C07305=1215.295,-74.617,-38.578,179.642,5.411,149.053
C07306=1215.289,-74.347,-38.590,179.644,5.412,149.052
C07307=1215.284,-74.097,-38.601,179.647,5.412,149.051
C07308=1215.278,-73.847,-38.613,179.649,5.412,149.051
C07309=1215.274,-73.598,-38.625,179.652,5.412,149.050
C07310=1215.268,-73.348,-38.636,179.653,5.412,149.049
C07311=1215.263,-73.098,-38.647,179.656,5.413,149.049
C07312=1215.258,-72.848,-38.658,179.658,5.413,149.048
C07313=1215.253,-72.599,-38.670,179.661,5.413,149.047
C07314=1215.247,-72.350,-38.681,179.663,5.413,149.047
C07315=1215.242,-72.100,-38.693,179.665,5.413,149.046
C07316=1215.237,-71.850,-38.704,179.668,5.414,149.045
C07317=1215.232,-71.600,-38.715,179.670,5.413,149.045
C07318=1215.227,-71.350,-38.726,179.673,5.414,149.044
C07319=1215.221,-71.101,-38.737,179.675,5.413,149.043
C07320=1215.216,-70.851,-38.749,179.677,5.414,149.043
C07321=1215.211,-70.601,-38.760,179.680,5.415,149.042
C07322=1215.206,-70.351,-38.772,179.682,5.414,149.041
C07323=1215.201,-70.103,-38.783,179.685,5.415,149.041
C07324=1215.195,-69.853,-38.795,179.687,5.414,149.040
C07325=1215.190,-69.603,-38.806,179.689,5.415,149.039
C07326=1215.185,-69.353,-38.818,179.691,5.414,149.038
C07327=1215.180,-69.103,-38.829,179.694,5.415,149.038
C07328=1215.174,-68.854,-38.840,179.697,5.415,149.037
C07329=1215.169,-68.604,-38.852,179.699,5.415,149.036
C07330=1215.164,-68.354,-38.864,179.701,5.416,149.036
C07331=1215.159,-68.104,-38.875,179.703,5.415,149.035
C07332=1215.154,-67.854,-38.887,179.706,5.416,149.034
C07333=1215.149,-67.605,-38.898,179.708,5.416,149.034
C07334=1215.143,-67.356,-38.910,179.711,5.416,149.033
C07335=1215.138,-67.106,-38.921,179.713,5.416,149.032
C07336=1215.133,-66.856,-38.933,179.715,5.416,149.032
C07337=1215.128,-66.606,-38.944,179.718,5.417,149.031
C07338=1215.123,-66.356,-38.956,179.720,5.416,149.030
C07339=1215.118,-66.107,-38.967,179.723,5.417,149.029
C07340=1215.112,-65.858,-38.979,179.725,5.416,149.029
C07341=1215.107,-65.608,-38.990,179.727,5.417,149.028
C07342=1215.102,-65.358,-39.002,179.730,5.418,149.028
C07343=1215.097,-65.108,-39.014,179.732,5.417,149.027
C07344=1215.092,-64.858,-39.025,179.734,5.418,149.026
C07345=1215.086,-64.609,-39.037,179.737,5.417,149.025
C07346=1215.082,-64.360,-39.049,179.739,5.418,149.025
C07347=1215.077,-64.110,-39.061,179.741,5.417,149.024
C07348=1215.071,-63.861,-39.072,179.744,5.418,149.023
C07349=1215.066,-63.611,-39.084,179.747,5.418,149.023
C07350=1215.060,-63.361,-39.096,179.749,5.418,149.022
C07351=1215.056,-63.111,-39.107,179.751,5.418,149.021
C07352=1215.050,-62.861,-39.119,179.753,5.418,149.020
C07353=1215.046,-62.612,-39.130,179.756,5.419,149.020
C07354=1215.040,-62.362,-39.142,179.758,5.419,149.019
C07355=1215.035,-62.112,-39.154,179.760,5.419,149.019
C07356=1215.030,-61.863,-39.166,179.763,5.420,149.018
C07357=1215.024,-61.614,-39.177,179.765,5.419,149.017
C07358=1215.019,-61.364,-39.189,179.768,5.420,149.016
C07359=1215.014,-61.114,-39.201,179.770,5.420,149.016
C07360=1215.009,-60.864,-39.212,179.773,5.420,149.015
C07361=1215.003,-60.614,-39.224,179.775,5.420,149.014
C07362=1214.999,-60.365,-39.236,179.777,5.420,149.014
C07363=1214.994,-60.115,-39.248,179.780,5.420,149.013
C07364=1214.988,-59.865,-39.260,179.783,5.421,149.012
C07365=1214.983,-59.616,-39.271,179.784,5.421,149.012
C07366=1214.978,-59.366,-39.283,179.787,5.421,149.011
C07367=1214.973,-59.116,-39.296,179.789,5.421,149.010
C07368=1214.968,-58.867,-39.307,179.792,5.421,149.010
C07369=1214.963,-58.617,-39.319,179.794,5.421,149.009
C07370=1214.957,-58.367,-39.331,179.796,5.421,149.008
C07371=1214.953,-58.118,-39.343,179.799,5.422,149.008
C07372=1214.948,-57.868,-39.355,179.801,5.422,149.007
C07373=1214.942,-57.618,-39.367,179.804,5.422,149.006
C07374=1214.937,-57.368,-39.378,179.806,5.422,149.005
C07375=1214.932,-57.119,-39.391,179.809,5.422,149.005
C07376=1214.927,-56.869,-39.402,179.811,5.423,149.004
C07377=1214.921,-56.620,-39.414,179.813,5.422,149.003
C07378=1214.916,-56.370,-39.425,179.816,5.423,149.003
C07379=1214.911,-56.121,-39.438,179.818,5.424,149.002
C07380=1214.906,-55.871,-39.450,179.820,5.423,149.001
C07381=1214.900,-55.621,-39.462,179.823,5.424,149.001
C07382=1214.896,-55.372,-39.474,179.825,5.423,149.000
C07383=1214.890,-55.122,-39.486,179.828,5.424,148.999
C07384=1214.885,-54.872,-39.497,179.830,5.424,148.999
C07385=1214.880,-54.622,-39.510,179.832,5.424,148.998
C07386=1214.876,-54.372,-39.522,179.835,5.424,148.997
C07387=1214.870,-54.123,-39.534,179.837,5.424,148.996
C07388=1214.865,-53.873,-39.546,179.840,5.425,148.996
C07389=1214.860,-53.623,-39.558,179.843,5.425,148.995
C07390=1214.855,-53.374,-39.571,179.845,5.425,148.994
C07391=1214.850,-53.124,-39.582,179.847,5.425,148.994
C07392=1214.844,-52.874,-39.594,179.849,5.425,148.993
C07393=1214.839,-52.625,-39.606,179.852,5.426,148.993
C07394=1214.834,-52.375,-39.618,179.854,5.426,148.992
C07395=1214.829,-52.126,-39.631,179.856,5.426,148.991
C07396=1214.824,-51.876,-39.642,179.859,5.426,148.990
C07397=1214.819,-51.627,-39.655,179.862,5.427,148.990
C07398=1214.814,-51.377,-39.667,179.864,5.426,148.989
C07399=1214.808,-51.127,-39.679,179.866,5.427,148.988
C07400=1214.803,-50.878,-39.691,179.868,5.426,148.988
C07401=1214.798,-50.628,-39.703,179.871,5.427,148.987
C07402=1214.792,-50.378,-39.716,179.874,5.427,148.986
C07403=1214.788,-50.129,-39.727,179.876,5.427,148.985
C07404=1214.783,-49.879,-39.740,179.879,5.428,148.985
C07405=1214.777,-49.630,-39.751,179.881,5.428,148.984
C07406=1214.773,-49.380,-39.764,179.883,5.428,148.984
C07407=1214.767,-49.110,-39.777,179.886,5.428,148.983
C07408=1214.761,-48.840,-39.790,179.889,5.429,148.982
C07409=1214.755,-48.570,-39.804,179.891,5.428,148.981
C07410=1214.750,-48.300,-39.817,179.893,5.429,148.981
C07411=1214.745,-48.051,-39.829,179.896,5.429,148.980
C07412=1214.739,-47.801,-39.841,179.898,5.429,148.979
C07413=1214.734,-47.551,-39.854,179.901,5.429,148.978
C07414=1214.729,-47.301,-39.866,179.903,5.430,148.978
C07415=1214.724,-47.051,-39.879,179.906,5.429,148.977
C07416=1214.719,-46.802,-39.891,179.908,5.430,148.976
C07417=1214.714,-46.552,-39.903,179.911,5.430,148.976
C07418=1214.709,-46.303,-39.915,179.913,5.430,148.975
C07419=1214.704,-46.053,-39.927,179.915,5.431,148.974
C07420=1214.699,-45.804,-39.940,179.918,5.431,148.974
C07421=1214.694,-45.554,-39.952,179.920,5.431,148.973
C07422=1214.688,-45.305,-39.964,179.923,5.431,148.972
C07423=1214.684,-45.055,-39.977,179.925,5.431,148.972
C07424=1214.678,-44.805,-39.989,179.927,5.432,148.971
C07425=1214.673,-44.555,-40.002,179.930,5.432,148.970
C07426=1214.668,-44.306,-40.014,179.932,5.432,148.970
C07427=1214.663,-44.056,-40.026,179.935,5.432,148.969
C07428=1214.657,-43.807,-40.039,179.937,5.433,148.968
C07429=1214.653,-43.557,-40.052,179.939,5.432,148.967
C07430=1214.647,-43.307,-40.064,179.942,5.433,148.967
C07431=1214.642,-43.057,-40.076,179.945,5.433,148.966
C07432=1214.637,-42.808,-40.089,179.947,5.433,148.965
C07433=1214.632,-42.558,-40.101,179.950,5.433,148.965
C07434=1214.627,-42.309,-40.113,179.952,5.434,148.964
C07435=1214.622,-42.059,-40.126,179.954,5.434,148.963
C07436=1214.617,-41.810,-40.139,179.956,5.434,148.963
C07437=1214.611,-41.559,-40.151,179.959,5.435,148.962
C07438=1214.606,-41.310,-40.164,179.961,5.435,148.961
C07439=1214.601,-41.061,-40.177,179.964,5.435,148.961
C07440=1214.596,-40.811,-40.190,179.966,5.435,148.960
C07441=1214.591,-40.561,-40.201,179.969,5.435,148.959
C07442=1214.585,-40.311,-40.214,179.971,5.436,148.959
C07443=1214.580,-40.062,-40.227,179.973,5.435,148.958
C07444=1214.575,-39.813,-40.239,179.976,5.436,148.957
C07445=1214.570,-39.562,-40.251,179.979,5.436,148.956
C07446=1214.565,-39.313,-40.264,179.981,5.436,148.956
C07447=1214.560,-39.063,-40.277,179.983,5.436,148.955
C07448=1214.555,-38.814,-40.289,179.986,5.437,148.954
C07449=1214.549,-38.565,-40.302,179.988,5.437,148.954
C07450=1214.544,-38.314,-40.315,179.990,5.437,148.953
C07451=1214.539,-38.065,-40.327,179.993,5.438,148.952
C07452=1214.534,-37.815,-40.340,179.995,5.438,148.952
C07453=1214.529,-37.566,-40.353,179.998,5.438,148.951
C07454=1214.524,-37.316,-40.366,-180.000,5.439,148.950
C07455=1214.519,-37.067,-40.378,-179.998,5.438,148.950
C07456=1214.513,-36.817,-40.391,-179.995,5.439,148.949
C07457=1214.508,-36.567,-40.403,-179.992,5.439,148.948
C07458=1214.504,-36.317,-40.416,-179.990,5.439,148.948
C07459=1214.498,-36.068,-40.429,-179.987,5.439,148.947
C07460=1214.493,-35.818,-40.441,-179.985,5.440,148.946
C07461=1214.488,-35.569,-40.454,-179.983,5.439,148.945
C07462=1214.483,-35.319,-40.468,-179.980,5.440,148.945
C07463=1214.478,-35.069,-40.480,-179.977,5.440,148.944
C07464=1214.473,-34.820,-40.493,-179.976,5.440,148.944
C07465=1214.468,-34.570,-40.506,-179.973,5.441,148.943
C07466=1214.463,-34.321,-40.518,-179.970,5.441,148.942
C07467=1214.457,-34.071,-40.531,-179.968,5.441,148.942
C07468=1214.452,-33.822,-40.544,-179.966,5.442,148.941
C07469=1214.447,-33.572,-40.557,-179.963,5.442,148.940
C07470=1214.442,-33.322,-40.569,-179.961,5.442,148.939
C07471=1214.436,-33.072,-40.582,-179.958,5.442,148.939
C07472=1214.432,-32.822,-40.595,-179.956,5.443,148.938
C07473=1214.427,-32.573,-40.608,-179.953,5.443,148.937
C07474=1214.421,-32.324,-40.620,-179.951,5.443,148.937
C07475=1214.416,-32.073,-40.634,-179.948,5.443,148.936
C07476=1214.411,-31.824,-40.646,-179.946,5.444,148.935
C07477=1214.406,-31.575,-40.660,-179.943,5.443,148.935
C07478=1214.402,-31.325,-40.673,-179.941,5.444,148.934
C07479=1214.396,-31.076,-40.686,-179.938,5.444,148.933
C07480=1214.391,-30.826,-40.699,-179.937,5.444,148.933
C07481=1214.386,-30.576,-40.712,-179.934,5.445,148.932
C07482=1214.381,-30.327,-40.724,-179.931,5.445,148.931
C07483=1214.375,-30.077,-40.737,-179.929,5.445,148.931
C07484=1214.371,-29.827,-40.750,-179.927,5.446,148.930
C07485=1214.366,-29.578,-40.763,-179.924,5.446,148.929
C07486=1214.360,-29.328,-40.776,-179.922,5.446,148.928
C07487=1214.355,-29.078,-40.789,-179.919,5.446,148.928
C07488=1214.350,-28.829,-40.802,-179.916,5.447,148.927
C07489=1214.345,-28.579,-40.815,-179.914,5.447,148.926
C07490=1214.340,-28.330,-40.829,-179.912,5.447,148.926
C07491=1214.335,-28.081,-40.841,-179.909,5.447,148.925
C07492=1214.330,-27.830,-40.855,-179.906,5.448,148.924
C07493=1214.324,-27.581,-40.867,-179.904,5.448,148.924
C07494=1214.319,-27.332,-40.880,-179.902,5.448,148.923
C07495=1214.314,-27.081,-40.893,-179.899,5.448,148.922
C07496=1214.309,-26.832,-40.906,-179.897,5.449,148.922
C07497=1214.305,-26.583,-40.920,-179.895,5.449,148.921
C07498=1214.299,-26.333,-40.933,-179.892,5.449,148.920
C07499=1214.294,-26.084,-40.946,-179.889,5.450,148.920
C07500=1214.288,-25.833,-40.959,-179.887,5.450,148.919
C07501=1214.283,-25.584,-40.972,-179.885,5.450,148.918
C07502=1214.279,-25.335,-40.985,-179.882,5.451,148.918
C07503=1214.273,-25.085,-40.999,-179.880,5.450,148.917
C07504=1214.269,-24.835,-41.012,-179.877,5.451,148.916
C07505=1214.263,-24.585,-41.025,-179.875,5.451,148.915
C07506=1214.258,-24.337,-41.038,-179.873,5.451,148.915
C07507=1214.254,-24.087,-41.051,-179.870,5.451,148.914
C07508=1214.248,-23.837,-41.064,-179.867,5.452,148.913
C07509=1214.243,-23.587,-41.077,-179.865,5.452,148.913
C07510=1214.238,-23.338,-41.091,-179.862,5.452,148.912
C07511=1214.233,-23.068,-41.105,-179.860,5.453,148.911
C07512=1214.227,-22.799,-41.120,-179.857,5.453,148.911
C07513=1214.221,-22.530,-41.134,-179.855,5.454,148.910
C07514=1214.216,-22.260,-41.148,-179.852,5.454,148.909
C07515=1214.211,-22.010,-41.162,-179.850,5.454,148.909
C07516=1214.206,-21.761,-41.174,-179.847,5.454,148.908
C07517=1214.200,-21.511,-41.187,-179.844,5.455,148.907
C07518=1214.196,-21.262,-41.201,-179.842,5.455,148.906
C07519=1214.190,-21.012,-41.214,-179.840,5.455,148.906
C07520=1214.186,-20.763,-41.228,-179.837,5.455,148.905
C07521=1214.180,-20.513,-41.241,-179.834,5.456,148.904
C07522=1214.175,-20.263,-41.254,-179.832,5.456,148.904
C07523=1214.170,-20.014,-41.268,-179.830,5.456,148.903
C07524=1214.165,-19.764,-41.281,-179.827,5.457,148.902
C07525=1214.159,-19.514,-41.294,-179.825,5.457,148.902
C07526=1214.155,-19.265,-41.308,-179.823,5.457,148.901
C07527=1214.149,-19.015,-41.321,-179.820,5.458,148.900
C07528=1214.145,-18.766,-41.335,-179.817,5.458,148.900
C07529=1214.139,-18.516,-41.348,-179.815,5.459,148.899
C07530=1214.135,-18.266,-41.361,-179.813,5.458,148.898
C07531=1214.129,-18.017,-41.375,-179.810,5.459,148.898
C07532=1214.124,-17.767,-41.388,-179.807,5.459,148.897
C07533=1214.119,-17.518,-41.402,-179.805,5.460,148.896
C07534=1214.114,-17.268,-41.415,-179.803,5.459,148.896
C07535=1214.110,-17.019,-41.429,-179.800,5.460,148.895
C07536=1214.104,-16.769,-41.442,-179.797,5.460,148.894
C07537=1214.099,-16.520,-41.456,-179.795,5.460,148.893
C07538=1214.094,-16.270,-41.469,-179.793,5.461,148.893
C07539=1214.089,-16.020,-41.483,-179.790,5.461,148.892
C07540=1214.083,-15.771,-41.496,-179.788,5.462,148.892
C07541=1214.079,-15.521,-41.510,-179.786,5.462,148.891
C07542=1214.073,-15.272,-41.523,-179.783,5.462,148.890
C07543=1214.068,-15.022,-41.537,-179.780,5.463,148.890
C07544=1214.063,-14.772,-41.551,-179.778,5.463,148.889
C07545=1214.058,-14.523,-41.564,-179.776,5.463,148.888
C07546=1214.053,-14.273,-41.578,-179.773,5.463,148.887
C07547=1214.048,-14.024,-41.591,-179.770,5.464,148.887
C07548=1214.043,-13.774,-41.604,-179.768,5.464,148.886
C07549=1214.037,-13.525,-41.618,-179.766,5.464,148.885
C07550=1214.033,-13.275,-41.633,-179.763,5.464,148.885
C07551=1214.028,-13.025,-41.646,-179.760,5.465,148.884
C07552=1214.022,-12.776,-41.659,-179.758,5.465,148.883
C07553=1214.017,-12.526,-41.673,-179.756,5.466,148.883
C07554=1214.012,-12.277,-41.686,-179.753,5.466,148.882
C07555=1214.007,-12.027,-41.701,-179.751,5.467,148.881
C07556=1214.002,-11.777,-41.714,-179.748,5.467,148.881
C07557=1213.997,-11.528,-41.727,-179.746,5.467,148.880
C07558=1213.992,-11.279,-41.742,-179.743,5.467,148.879
C07559=1213.987,-11.029,-41.755,-179.741,5.468,148.879
C07560=1213.982,-10.779,-41.769,-179.738,5.468,148.878
C07561=1213.977,-10.530,-41.783,-179.736,5.468,148.877
C07562=1213.971,-10.280,-41.796,-179.733,5.468,148.877
C07563=1213.967,-10.030,-41.810,-179.731,5.469,148.876
C07564=1213.962,-9.781,-41.824,-179.728,5.469,148.875
C07565=1213.956,-9.531,-41.837,-179.725,5.470,148.875
C07566=1213.951,-9.282,-41.852,-179.723,5.470,148.874
C07567=1213.947,-9.032,-41.866,-179.721,5.470,148.873
C07568=1213.941,-8.783,-41.878,-179.718,5.471,148.873
C07569=1213.936,-8.533,-41.893,-179.716,5.471,148.872
C07570=1213.932,-8.283,-41.907,-179.714,5.471,148.871
C07571=1213.926,-8.034,-41.921,-179.711,5.472,148.871
C07572=1213.921,-7.784,-41.934,-179.708,5.472,148.870
C07573=1213.916,-7.535,-41.948,-179.706,5.473,148.869
C07574=1213.911,-7.286,-41.962,-179.704,5.472,148.869
C07575=1213.906,-7.036,-41.976,-179.701,5.473,148.868
C07576=1213.901,-6.785,-41.990,-179.698,5.473,148.867
C07577=1213.896,-6.537,-42.003,-179.696,5.474,148.866
C07578=1213.891,-6.287,-42.017,-179.693,5.474,148.866
C07579=1213.886,-6.037,-42.032,-179.691,5.474,148.865
C07580=1213.881,-5.788,-42.046,-179.689,5.475,148.865
C07581=1213.875,-5.539,-42.060,-179.686,5.475,148.864
C07582=1213.870,-5.288,-42.074,-179.683,5.476,148.863
C07583=1213.866,-5.039,-42.087,-179.681,5.476,148.863
C07584=1213.860,-4.790,-42.101,-179.679,5.476,148.862
C07585=1213.855,-4.540,-42.115,-179.676,5.477,148.861
C07586=1213.851,-4.290,-42.130,-179.673,5.477,148.860
C07587=1213.845,-4.041,-42.144,-179.671,5.478,148.860
C07588=1213.840,-3.792,-42.158,-179.669,5.477,148.859
C07589=1213.835,-3.541,-42.171,-179.666,5.478,148.858
C07590=1213.831,-3.292,-42.185,-179.663,5.478,148.858
C07591=1213.825,-3.043,-42.199,-179.661,5.479,148.857
C07592=1213.820,-2.793,-42.213,-179.659,5.480,148.857
C07593=1213.815,-2.544,-42.228,-179.657,5.479,148.856
C07594=1213.810,-2.294,-42.242,-179.654,5.480,148.855
C07595=1213.805,-2.045,-42.256,-179.651,5.480,148.854
C07596=1213.800,-1.795,-42.270,-179.649,5.481,148.854
C07597=1213.795,-1.545,-42.284,-179.646,5.481,148.853
C07598=1213.790,-1.296,-42.299,-179.644,5.481,148.852
C07599=1213.784,-1.047,-42.312,-179.641,5.482,148.852
C07600=1213.779,-0.797,-42.327,-179.639,5.482,148.851
C07601=1213.775,-0.548,-42.340,-179.636,5.483,148.850
C07602=1213.770,-0.298,-42.355,-179.633,5.483,148.850
C07603=1213.765,-0.048,-42.369,-179.631,5.483,148.849
C07604=1213.760,0.201,-42.383,-179.629,5.484,148.849
C07605=1213.755,0.451,-42.397,-179.626,5.484,148.848
C07606=1213.750,0.700,-42.411,-179.624,5.485,148.847
C07607=1213.745,0.950,-42.426,-179.621,5.485,148.846
C07608=1213.740,1.200,-42.440,-179.619,5.485,148.846
C07609=1213.734,1.449,-42.454,-179.616,5.485,148.845
C07610=1213.729,1.698,-42.468,-179.614,5.486,148.844
C07611=1213.724,1.948,-42.482,-179.611,5.486,148.844
C07612=1213.719,2.198,-42.497,-179.608,5.487,148.843
C07613=1213.714,2.448,-42.511,-179.606,5.487,148.842
C07614=1213.709,2.697,-42.525,-179.604,5.487,148.842
C07615=1213.704,2.965,-42.541,-179.601,5.488,148.841
C07616=1213.698,3.235,-42.556,-179.598,5.488,148.840
C07617=1213.692,3.504,-42.572,-179.596,5.489,148.840
C07618=1213.687,3.773,-42.587,-179.593,5.489,148.839
C07619=1213.682,4.023,-42.601,-179.590,5.490,148.838
C07620=1213.677,4.272,-42.616,-179.588,5.490,148.838
C07621=1213.672,4.521,-42.630,-179.585,5.491,148.837
C07622=1213.667,4.771,-42.644,-179.583,5.490,148.836
C07623=1213.662,5.020,-42.659,-179.580,5.491,148.835
C07624=1213.657,5.270,-42.673,-179.578,5.491,148.835
C07625=1213.652,5.520,-42.687,-179.575,5.492,148.834
C07626=1213.647,5.769,-42.702,-179.573,5.493,148.834
C07627=1213.642,6.019,-42.717,-179.571,5.493,148.833
C07628=1213.637,6.268,-42.730,-179.568,5.493,148.832
C07629=1213.631,6.518,-42.745,-179.565,5.494,148.832
C07630=1213.626,6.767,-42.760,-179.563,5.494,148.831
C07631=1213.621,7.017,-42.775,-179.560,5.495,148.830
C07632=1213.617,7.266,-42.789,-179.557,5.495,148.829
C07633=1213.612,7.516,-42.803,-179.555,5.495,148.829
C07634=1213.607,7.766,-42.817,-179.553,5.495,148.828
C07635=1213.602,8.015,-42.832,-179.551,5.496,148.828
C07636=1213.597,8.264,-42.847,-179.548,5.497,148.827
C07637=1213.592,8.514,-42.861,-179.545,5.497,148.826
C07638=1213.586,8.763,-42.875,-179.543,5.498,148.826
C07639=1213.581,9.013,-42.890,-179.541,5.497,148.825
C07640=1213.576,9.262,-42.905,-179.538,5.498,148.824
C07641=1213.571,9.512,-42.919,-179.535,5.499,148.824
C07642=1213.567,9.761,-42.934,-179.533,5.499,148.823
C07643=1213.562,10.011,-42.948,-179.530,5.500,148.822
C07644=1213.556,10.261,-42.963,-179.527,5.500,148.821
C07645=1213.551,10.511,-42.977,-179.525,5.501,148.821
C07646=1213.546,10.760,-42.992,-179.523,5.501,148.820
C07647=1213.541,11.009,-43.007,-179.520,5.501,148.820
C07648=1213.537,11.258,-43.022,-179.518,5.502,148.819
C07649=1213.531,11.508,-43.037,-179.515,5.502,148.818
C07650=1213.526,11.758,-43.051,-179.512,5.503,148.818
C07651=1213.521,12.007,-43.066,-179.510,5.503,148.817
C07652=1213.516,12.257,-43.080,-179.507,5.504,148.816
C07653=1213.511,12.507,-43.095,-179.505,5.503,148.816
C07654=1213.506,12.756,-43.110,-179.503,5.504,148.815
C07655=1213.501,13.006,-43.124,-179.500,5.505,148.814
C07656=1213.496,13.255,-43.139,-179.498,5.505,148.814
C07657=1213.491,13.505,-43.154,-179.495,5.506,148.813
C07658=1213.486,13.755,-43.168,-179.492,5.506,148.812
C07659=1213.481,14.004,-43.183,-179.490,5.507,148.812
C07660=1213.476,14.253,-43.198,-179.488,5.507,148.811
C07661=1213.471,14.503,-43.213,-179.485,5.507,148.810
C07662=1213.466,14.753,-43.228,-179.482,5.508,148.810
C07663=1213.461,15.002,-43.243,-179.480,5.509,148.809
C07664=1213.456,15.252,-43.257,-179.478,5.509,148.808
C07665=1213.451,15.501,-43.272,-179.475,5.510,148.808
C07666=1213.446,15.750,-43.287,-179.472,5.510,148.807
C07667=1213.441,16.000,-43.302,-179.470,5.510,148.806
C07668=1213.436,16.250,-43.317,-179.468,5.510,148.806
C07669=1213.431,16.499,-43.332,-179.465,5.511,148.805
C07670=1213.426,16.748,-43.346,-179.462,5.511,148.804
C07671=1213.421,16.998,-43.361,-179.460,5.512,148.804
C07672=1213.416,17.247,-43.376,-179.457,5.513,148.803
C07673=1213.411,17.497,-43.391,-179.455,5.513,148.803
C07674=1213.406,17.746,-43.406,-179.452,5.514,148.802
C07675=1213.401,17.996,-43.421,-179.450,5.514,148.801
C07676=1213.395,18.245,-43.436,-179.447,5.514,148.801
C07677=1213.390,18.495,-43.450,-179.445,5.515,148.800
C07678=1213.386,18.744,-43.465,-179.442,5.515,148.799
C07679=1213.380,18.994,-43.480,-179.439,5.516,148.798
C07680=1213.375,19.243,-43.495,-179.437,5.517,148.798
C07681=1213.371,19.492,-43.510,-179.435,5.517,148.797
C07682=1213.365,19.742,-43.525,-179.432,5.518,148.797
C07683=1213.360,19.991,-43.540,-179.429,5.518,148.796
C07684=1213.356,20.241,-43.556,-179.427,5.518,148.795
C07685=1213.351,20.491,-43.570,-179.425,5.518,148.795
C07686=1213.346,20.740,-43.585,-179.422,5.519,148.794
C07687=1213.341,20.990,-43.601,-179.419,5.519,148.793
C07688=1213.336,21.239,-43.615,-179.417,5.520,148.793
C07689=1213.330,21.489,-43.631,-179.415,5.521,148.792
C07690=1213.326,21.738,-43.646,-179.412,5.521,148.791
C07691=1213.320,21.988,-43.661,-179.409,5.522,148.791
C07692=1213.315,22.237,-43.676,-179.407,5.522,148.790
C07693=1213.310,22.486,-43.691,-179.405,5.522,148.789
C07694=1213.306,22.736,-43.707,-179.402,5.523,148.789
C07695=1213.300,22.986,-43.721,-179.399,5.523,148.788
C07696=1213.295,23.235,-43.736,-179.397,5.524,148.788
C07697=1213.290,23.485,-43.752,-179.394,5.525,148.787
C07698=1213.285,23.734,-43.767,-179.392,5.525,148.786
C07699=1213.280,23.984,-43.782,-179.389,5.526,148.786
C07700=1213.275,24.233,-43.797,-179.387,5.526,148.785
C07701=1213.270,24.483,-43.813,-179.384,5.527,148.784
C07702=1213.266,24.732,-43.828,-179.381,5.527,148.784
C07703=1213.260,24.982,-43.843,-179.379,5.528,148.783
C07704=1213.255,25.231,-43.858,-179.377,5.528,148.782
C07705=1213.250,25.480,-43.873,-179.374,5.528,148.782
C07706=1213.245,25.730,-43.888,-179.372,5.529,148.781
C07707=1213.240,25.980,-43.904,-179.369,5.529,148.780
C07708=1213.236,26.229,-43.919,-179.366,5.530,148.780
C07709=1213.230,26.479,-43.934,-179.364,5.531,148.779
C07710=1213.225,26.728,-43.949,-179.361,5.531,148.778
C07711=1213.220,26.977,-43.965,-179.359,5.532,148.778
C07712=1213.215,27.226,-43.980,-179.356,5.532,148.777
C07713=1213.211,27.476,-43.996,-179.354,5.533,148.776
C07714=1213.205,27.726,-44.011,-179.351,5.534,148.776
C07715=1213.201,27.975,-44.026,-179.348,5.534,148.775
C07716=1213.195,28.224,-44.042,-179.346,5.534,148.774
C07717=1213.191,28.473,-44.057,-179.344,5.534,148.774
C07718=1213.186,28.724,-44.072,-179.342,5.535,148.773
C07719=1213.180,28.993,-44.089,-179.338,5.535,148.772
C07720=1213.175,29.261,-44.105,-179.336,5.536,148.772
C07721=1213.169,29.530,-44.122,-179.333,5.537,148.771
C07722=1213.164,29.798,-44.139,-179.330,5.538,148.770
C07723=1213.159,30.047,-44.154,-179.327,5.538,148.770
C07724=1213.154,30.298,-44.170,-179.326,5.538,148.769
C07725=1213.149,30.547,-44.185,-179.323,5.539,148.769
C07726=1213.144,30.796,-44.200,-179.320,5.539,148.768
C07727=1213.139,31.045,-44.216,-179.318,5.540,148.767
C07728=1213.133,31.295,-44.231,-179.315,5.541,148.767
C07729=1213.129,31.545,-44.247,-179.312,5.541,148.766
C07730=1213.124,31.794,-44.262,-179.310,5.542,148.765
C07731=1213.119,32.043,-44.278,-179.308,5.542,148.765
C07732=1213.115,32.293,-44.293,-179.305,5.543,148.764
C07733=1213.109,32.543,-44.309,-179.302,5.544,148.763
C07734=1213.104,32.792,-44.325,-179.300,5.544,148.763
C07735=1213.099,33.041,-44.340,-179.297,5.545,148.762
C07736=1213.094,33.291,-44.355,-179.294,5.545,148.761
C07737=1213.089,33.541,-44.371,-179.292,5.546,148.761
C07738=1213.084,33.790,-44.387,-179.290,5.547,148.760
C07739=1213.080,34.039,-44.403,-179.287,5.547,148.760
C07740=1213.074,34.289,-44.418,-179.284,5.548,148.759
C07741=1213.069,34.538,-44.434,-179.282,5.548,148.758
C07742=1213.064,34.787,-44.450,-179.279,5.549,148.758
C07743=1213.060,35.037,-44.465,-179.277,5.549,148.757
C07744=1213.054,35.287,-44.480,-179.275,5.549,148.756
C07745=1213.049,35.536,-44.496,-179.272,5.550,148.756
C07746=1213.044,35.786,-44.512,-179.270,5.550,148.755
C07747=1213.040,36.035,-44.528,-179.267,5.551,148.754
C07748=1213.034,36.284,-44.543,-179.264,5.552,148.754
C07749=1213.030,36.534,-44.559,-179.262,5.552,148.753
C07750=1213.024,36.784,-44.575,-179.259,5.553,148.753
C07751=1213.019,37.033,-44.590,-179.257,5.554,148.752
C07752=1213.015,37.282,-44.606,-179.254,5.554,148.751
C07753=1213.010,37.532,-44.622,-179.252,5.555,148.751
C07754=1213.004,37.781,-44.638,-179.249,5.555,148.750
C07755=1213.000,38.031,-44.654,-179.247,5.556,148.749
C07756=1212.994,38.280,-44.669,-179.244,5.557,148.749
C07757=1212.989,38.529,-44.686,-179.241,5.557,148.748
C07758=1212.985,38.779,-44.701,-179.239,5.558,148.747
C07759=1212.980,39.028,-44.716,-179.236,5.558,148.747
C07760=1212.975,39.278,-44.733,-179.234,5.559,148.746
C07761=1212.970,39.527,-44.749,-179.231,5.560,148.746
C07762=1212.964,39.777,-44.764,-179.229,5.560,148.745
C07763=1212.960,40.027,-44.780,-179.226,5.561,148.744
C07764=1212.954,40.276,-44.797,-179.223,5.561,148.744
C07765=1212.949,40.525,-44.812,-179.221,5.562,148.743
C07766=1212.945,40.775,-44.828,-179.218,5.562,148.742
C07767=1212.940,41.024,-44.844,-179.216,5.563,148.742
C07768=1212.935,41.274,-44.860,-179.213,5.564,148.741
C07769=1212.930,41.523,-44.875,-179.211,5.564,148.740
C07770=1212.925,41.772,-44.892,-179.208,5.565,148.740
C07771=1212.920,42.022,-44.908,-179.205,5.565,148.739
C07772=1212.915,42.271,-44.923,-179.203,5.566,148.739
C07773=1212.910,42.521,-44.940,-179.201,5.567,148.738
C07774=1212.905,42.770,-44.955,-179.198,5.567,148.737
C07775=1212.900,43.020,-44.972,-179.195,5.568,148.737
C07776=1212.895,43.269,-44.988,-179.193,5.568,148.736
C07777=1212.889,43.519,-45.003,-179.190,5.569,148.735
C07778=1212.885,43.768,-45.020,-179.188,5.570,148.735
C07779=1212.880,44.017,-45.036,-179.185,5.570,148.734
C07780=1212.876,44.267,-45.052,-179.183,5.571,148.734
C07781=1212.870,44.516,-45.067,-179.180,5.572,148.733
C07782=1212.866,44.765,-45.084,-179.177,5.572,148.732
C07783=1212.861,45.015,-45.099,-179.175,5.573,148.732
C07784=1212.856,45.264,-45.116,-179.173,5.574,148.731
C07785=1212.851,45.514,-45.132,-179.170,5.574,148.730
C07786=1212.846,45.763,-45.148,-179.167,5.575,148.730
C07787=1212.841,46.013,-45.164,-179.165,5.575,148.729
C07788=1212.836,46.262,-45.181,-179.163,5.576,148.729
C07789=1212.831,46.512,-45.196,-179.160,5.577,148.728
C07790=1212.826,46.761,-45.214,-179.157,5.577,148.727
C07791=1212.820,47.011,-45.229,-179.155,5.578,148.727
C07792=1212.815,47.259,-45.245,-179.152,5.578,148.726
C07793=1212.810,47.510,-45.261,-179.150,5.579,148.725
C07794=1212.806,47.759,-45.278,-179.147,5.580,148.725
C07795=1212.801,48.008,-45.294,-179.145,5.580,148.724
C07796=1212.796,48.258,-45.310,-179.142,5.581,148.723
C07797=1212.791,48.507,-45.327,-179.139,5.581,148.723
C07798=1212.786,48.757,-45.343,-179.137,5.582,148.722
C07799=1212.781,49.006,-45.359,-179.135,5.583,148.722
C07800=1212.776,49.256,-45.375,-179.132,5.583,148.721
C07801=1212.771,49.505,-45.391,-179.129,5.584,148.720
C07802=1212.767,49.754,-45.408,-179.127,5.585,148.720
C07803=1212.761,50.003,-45.423,-179.125,5.585,148.719
C07804=1212.756,50.253,-45.441,-179.122,5.586,148.719
C07805=1212.751,50.502,-45.457,-179.119,5.587,148.718
C07806=1212.746,50.752,-45.473,-179.117,5.587,148.717
C07807=1212.741,51.001,-45.489,-179.114,5.588,148.717
C07808=1212.737,51.250,-45.506,-179.112,5.589,148.716
C07809=1212.732,51.500,-45.522,-179.109,5.589,148.715
C07810=1212.727,51.749,-45.538,-179.107,5.590,148.715
C07811=1212.722,51.999,-45.555,-179.104,5.590,148.714
C07812=1212.717,52.248,-45.572,-179.101,5.591,148.713
C07813=1212.712,52.498,-45.588,-179.099,5.592,148.713
C07814=1212.707,52.747,-45.604,-179.096,5.592,148.712
C07815=1212.702,52.996,-45.621,-179.093,5.594,148.712
C07816=1212.698,53.246,-45.637,-179.091,5.594,148.711
C07817=1212.692,53.495,-45.653,-179.088,5.595,148.711
C07818=1212.687,53.745,-45.670,-179.086,5.596,148.710
C07819=1212.682,53.994,-45.686,-179.083,5.596,148.709
C07820=1212.678,54.243,-45.703,-179.081,5.597,148.709
C07821=1212.673,54.493,-45.719,-179.078,5.597,148.708
C07822=1212.667,54.742,-45.736,-179.076,5.598,148.707
C07823=1212.662,55.011,-45.754,-179.073,5.599,148.707
C07824=1212.657,55.279,-45.771,-179.071,5.599,148.706
C07825=1212.652,55.548,-45.789,-179.067,5.601,148.705
C07826=1212.646,55.816,-45.807,-179.065,5.601,148.705
C07827=1212.642,56.066,-45.824,-179.062,5.602,148.704
C07828=1212.636,56.315,-45.840,-179.059,5.602,148.703
C07829=1212.631,56.565,-45.857,-179.057,5.603,148.703
C07830=1212.627,56.814,-45.874,-179.055,5.604,148.702
C07831=1212.622,57.063,-45.890,-179.052,5.604,148.702
C07832=1212.617,57.313,-45.907,-179.049,5.605,148.701
C07833=1212.611,57.562,-45.924,-179.047,5.605,148.700
C07834=1212.607,57.811,-45.940,-179.045,5.606,148.700
C07835=1212.602,58.061,-45.957,-179.042,5.607,148.699
C07836=1212.596,58.310,-45.974,-179.039,5.607,148.699
C07837=1212.592,58.559,-45.990,-179.037,5.608,148.698
C07838=1212.587,58.809,-46.006,-179.034,5.610,148.698
C07839=1212.582,59.059,-46.024,-179.031,5.610,148.697
C07840=1212.577,59.308,-46.040,-179.029,5.611,148.696
C07841=1212.572,59.557,-46.057,-179.026,5.611,148.696
C07842=1212.567,59.807,-46.074,-179.023,5.612,148.695
C07843=1212.562,60.056,-46.090,-179.021,5.613,148.694
C07844=1212.558,60.305,-46.107,-179.019,5.613,148.694
C07845=1212.552,60.555,-46.124,-179.016,5.614,148.693
C07846=1212.547,60.804,-46.140,-179.013,5.615,148.692
C07847=1212.543,61.053,-46.157,-179.011,5.616,148.692
C07848=1212.538,61.303,-46.174,-179.009,5.616,148.691
C07849=1212.533,61.553,-46.191,-179.006,5.617,148.691
C07850=1212.527,61.802,-46.208,-179.003,5.618,148.690
C07851=1212.523,62.051,-46.225,-179.001,5.619,148.690
C07852=1212.519,62.300,-46.242,-178.998,5.619,148.689
C07853=1212.513,62.549,-46.259,-178.995,5.620,148.688
C07854=1212.508,62.799,-46.276,-178.993,5.621,148.688
C07855=1212.503,63.049,-46.293,-178.991,5.622,148.687
C07856=1212.499,63.298,-46.310,-178.988,5.622,148.686
C07857=1212.494,63.547,-46.326,-178.985,5.623,148.686
C07858=1212.488,63.797,-46.343,-178.983,5.623,148.685
C07859=1212.484,64.046,-46.360,-178.981,5.624,148.685
C07860=1212.479,64.296,-46.377,-178.978,5.625,148.684
C07861=1212.474,64.544,-46.394,-178.975,5.626,148.683
C07862=1212.469,64.794,-46.411,-178.973,5.627,148.683
C07863=1212.464,65.043,-46.428,-178.970,5.628,148.682
C07864=1212.459,65.293,-46.445,-178.967,5.628,148.682
C07865=1212.455,65.543,-46.462,-178.965,5.629,148.681
C07866=1212.449,65.792,-46.479,-178.963,5.630,148.681
C07867=1212.445,66.041,-46.496,-178.960,5.630,148.680
C07868=1212.439,66.290,-46.513,-178.957,5.631,148.679
C07869=1212.435,66.540,-46.530,-178.955,5.631,148.679
C07870=1212.430,66.790,-46.547,-178.952,5.633,148.678
C07871=1212.425,67.038,-46.564,-178.949,5.634,148.677
C07872=1212.420,67.288,-46.582,-178.947,5.634,148.677
C07873=1212.415,67.537,-46.598,-178.944,5.635,148.676
C07874=1212.410,67.787,-46.616,-178.942,5.636,148.676
C07875=1212.405,68.036,-46.632,-178.939,5.636,148.675
C07876=1212.401,68.286,-46.650,-178.937,5.637,148.674
C07877=1212.395,68.534,-46.667,-178.935,5.638,148.674
C07878=1212.390,68.784,-46.684,-178.931,5.639,148.673
C07879=1212.386,69.033,-46.701,-178.929,5.640,148.673
C07880=1212.381,69.283,-46.718,-178.926,5.640,148.672
C07881=1212.376,69.533,-46.736,-178.924,5.641,148.672
C07882=1212.371,69.781,-46.753,-178.921,5.642,148.671
C07883=1212.366,70.031,-46.770,-178.919,5.642,148.670
C07884=1212.361,70.280,-46.787,-178.917,5.643,148.670
C07885=1212.356,70.529,-46.805,-178.914,5.644,148.669
C07886=1212.351,70.779,-46.822,-178.911,5.645,148.668
C07887=1212.347,71.029,-46.839,-178.908,5.646,148.668
C07888=1212.342,71.278,-46.857,-178.906,5.647,148.667
C07889=1212.336,71.527,-46.874,-178.903,5.647,148.667
C07890=1212.332,71.776,-46.891,-178.901,5.648,148.666
C07891=1212.326,72.025,-46.908,-178.899,5.649,148.666
C07892=1212.322,72.275,-46.925,-178.896,5.649,148.665
C07893=1212.317,72.524,-46.943,-178.893,5.651,148.664
C07894=1212.312,72.774,-46.960,-178.890,5.651,148.664
C07895=1212.308,73.023,-46.977,-178.888,5.652,148.663
C07896=1212.302,73.273,-46.995,-178.885,5.653,148.663
C07897=1212.298,73.522,-47.013,-178.883,5.653,148.662
C07898=1212.293,73.771,-47.029,-178.881,5.654,148.661
C07899=1212.288,74.020,-47.047,-178.878,5.655,148.661
C07900=1212.283,74.270,-47.065,-178.875,5.656,148.660
C07901=1212.278,74.520,-47.082,-178.872,5.657,148.659
C07902=1212.273,74.768,-47.099,-178.870,5.658,148.659
C07903=1212.268,75.017,-47.117,-178.867,5.658,148.658
C07904=1212.263,75.267,-47.134,-178.865,5.659,148.658
C07905=1212.259,75.516,-47.151,-178.863,5.660,148.657
C07906=1212.253,75.766,-47.169,-178.859,5.661,148.657
C07907=1212.248,76.015,-47.187,-178.857,5.662,148.656
C07908=1212.243,76.265,-47.204,-178.855,5.663,148.656
C07909=1212.239,76.514,-47.221,-178.852,5.663,148.655
C07910=1212.234,76.763,-47.239,-178.849,5.664,148.654
C07911=1212.229,77.013,-47.257,-178.847,5.665,148.654
C07912=1212.224,77.262,-47.275,-178.844,5.666,148.653
C07913=1212.220,77.511,-47.291,-178.841,5.667,148.653
C07914=1212.215,77.760,-47.309,-178.839,5.667,148.652
C07915=1212.209,78.010,-47.327,-178.837,5.668,148.651
C07916=1212.205,78.259,-47.344,-178.834,5.669,148.651
C07917=1212.200,78.509,-47.362,-178.831,5.669,148.650
C07918=1212.195,78.758,-47.379,-178.829,5.671,148.650
C07919=1212.190,79.007,-47.397,-178.826,5.672,148.649
C07920=1212.185,79.256,-47.415,-178.823,5.672,148.648
C07921=1212.180,79.506,-47.432,-178.821,5.673,148.648
C07922=1212.175,79.755,-47.450,-178.819,5.674,148.647
C07923=1212.170,80.005,-47.468,-178.815,5.675,148.647
C07924=1212.166,80.254,-47.485,-178.813,5.676,148.646
C07925=1212.161,80.503,-47.503,-178.811,5.677,148.646
C07926=1212.156,80.752,-47.521,-178.808,5.677,148.645
C07927=1212.151,81.021,-47.540,-178.805,5.678,148.644
C07928=1212.145,81.290,-47.559,-178.803,5.679,148.644
C07929=1212.140,81.558,-47.578,-178.800,5.680,148.643
C07930=1212.134,81.826,-47.597,-178.797,5.681,148.643
C07931=1212.130,82.076,-47.615,-178.794,5.682,148.642
C07932=1212.125,82.325,-47.633,-178.792,5.683,148.641
C07933=1212.120,82.574,-47.651,-178.789,5.684,148.641
C07934=1212.115,82.824,-47.668,-178.787,5.684,148.640
C07935=1212.110,83.073,-47.686,-178.784,5.686,148.640
C07936=1212.105,83.322,-47.704,-178.782,5.686,148.639
C07937=1212.101,83.571,-47.722,-178.779,5.687,148.638
C07938=1212.096,83.820,-47.740,-178.777,5.688,148.638
C07939=1212.091,84.070,-47.758,-178.774,5.689,148.637
C07940=1212.086,84.319,-47.775,-178.771,5.690,148.637
C07941=1212.081,84.568,-47.793,-178.769,5.691,148.636
C07942=1212.076,84.818,-47.811,-178.766,5.691,148.636
C07943=1212.071,85.067,-47.829,-178.764,5.692,148.635
C07944=1212.066,85.316,-47.847,-178.761,5.693,148.635
C07945=1212.062,85.566,-47.865,-178.758,5.694,148.634
C07946=1212.057,85.815,-47.883,-178.756,5.695,148.633
C07947=1212.052,86.064,-47.901,-178.753,5.696,148.633
C07948=1212.047,86.314,-47.918,-178.751,5.696,148.632
C07949=1212.042,86.563,-47.936,-178.748,5.698,148.632
C07950=1212.037,86.812,-47.954,-178.746,5.699,148.631
C07951=1212.032,87.062,-47.972,-178.743,5.699,148.630
C07952=1212.027,87.311,-47.990,-178.740,5.700,148.630
C07953=1212.023,87.561,-48.009,-178.738,5.701,148.629
C07954=1212.018,87.810,-48.027,-178.735,5.702,148.629
C07955=1212.013,88.059,-48.045,-178.732,5.703,148.628
C07956=1212.008,88.308,-48.063,-178.730,5.704,148.628
C07957=1212.003,88.557,-48.081,-178.728,5.704,148.627
C07958=1211.999,88.806,-48.099,-178.725,5.706,148.627
C07959=1211.994,89.056,-48.117,-178.722,5.707,148.626
C07960=1211.989,89.306,-48.136,-178.720,5.707,148.625
C07961=1211.984,89.555,-48.153,-178.718,5.708,148.625
C07962=1211.979,89.804,-48.171,-178.714,5.710,148.624
C07963=1211.974,90.053,-48.189,-178.712,5.710,148.624
C07964=1211.969,90.303,-48.207,-178.710,5.711,148.623
C07965=1211.965,90.552,-48.226,-178.707,5.712,148.622
C07966=1211.960,90.801,-48.244,-178.704,5.713,148.622
C07967=1211.955,91.050,-48.262,-178.702,5.714,148.621
C07968=1211.950,91.299,-48.280,-178.699,5.715,148.621
C07969=1211.945,91.549,-48.299,-178.697,5.716,148.620
C07970=1211.940,91.799,-48.317,-178.694,5.717,148.620
C07971=1211.935,92.048,-48.335,-178.691,5.718,148.619
C07972=1211.930,92.297,-48.353,-178.689,5.719,148.619
C07973=1211.925,92.546,-48.371,-178.686,5.719,148.618
C07974=1211.921,92.795,-48.390,-178.684,5.721,148.618
C07975=1211.917,93.045,-48.408,-178.681,5.721,148.617
C07976=1211.911,93.294,-48.427,-178.678,5.722,148.616
C07977=1211.906,93.543,-48.445,-178.676,5.723,148.616
C07978=1211.901,93.793,-48.463,-178.673,5.724,148.615
C07979=1211.897,94.042,-48.482,-178.670,5.725,148.615
C07980=1211.892,94.291,-48.500,-178.668,5.726,148.614
C07981=1211.887,94.540,-48.518,-178.666,5.726,148.613
C07982=1211.882,94.790,-48.536,-178.663,5.728,148.613
C07983=1211.877,95.039,-48.555,-178.660,5.729,148.612
C07984=1211.873,95.288,-48.573,-178.658,5.729,148.612
C07985=1211.868,95.537,-48.591,-178.656,5.730,148.611
C07986=1211.862,95.787,-48.610,-178.652,5.732,148.611
C07987=1211.858,96.037,-48.628,-178.650,5.733,148.610
C07988=1211.853,96.285,-48.647,-178.648,5.733,148.610
C07989=1211.848,96.534,-48.665,-178.644,5.735,148.609
C07990=1211.843,96.784,-48.684,-178.642,5.736,148.609
C07991=1211.839,97.033,-48.703,-178.640,5.736,148.608
C07992=1211.834,97.282,-48.721,-178.638,5.737,148.608
C07993=1211.828,97.532,-48.739,-178.634,5.739,148.607
C07994=1211.824,97.781,-48.758,-178.632,5.739,148.606
C07995=1211.819,98.030,-48.776,-178.630,5.740,148.606
C07996=1211.814,98.279,-48.794,-178.626,5.742,148.605
C07997=1211.809,98.529,-48.814,-178.624,5.742,148.605
C07998=1211.805,98.778,-48.832,-178.622,5.743,148.604
C07999=1211.800,99.027,-48.850,-178.619,5.744,148.603
C08000=1211.795,99.277,-48.870,-178.616,5.745,148.603
C08001=1211.790,99.526,-48.888,-178.614,5.746,148.602
C08002=1211.785,99.775,-48.906,-178.612,5.747,148.602
C08003=1211.780,100.025,-48.925,-178.608,5.748,148.601
C08004=1211.776,100.273,-48.944,-178.606,5.749,148.601
C08005=1211.771,100.522,-48.962,-178.604,5.750,148.600
C08006=1211.766,100.773,-48.981,-178.601,5.751,148.600
C08007=1211.761,101.021,-48.999,-178.598,5.752,148.599
C08008=1211.756,101.271,-49.018,-178.596,5.753,148.599
C08009=1211.752,101.520,-49.037,-178.594,5.754,148.598
C08010=1211.747,101.769,-49.055,-178.590,5.755,148.598
C08011=1211.741,102.018,-49.074,-178.588,5.756,148.597
C08012=1211.737,102.268,-49.093,-178.586,5.757,148.596
C08013=1211.732,102.517,-49.112,-178.583,5.758,148.596
C08014=1211.727,102.767,-49.130,-178.580,5.759,148.595
C08015=1211.723,103.015,-49.149,-178.578,5.760,148.595
C08016=1211.717,103.265,-49.168,-178.575,5.761,148.594
C08017=1211.713,103.514,-49.187,-178.572,5.762,148.594
C08018=1211.708,103.763,-49.206,-178.570,5.763,148.593
C08019=1211.703,104.013,-49.224,-178.567,5.764,148.593
C08020=1211.698,104.262,-49.244,-178.565,5.765,148.592
C08021=1211.693,104.511,-49.262,-178.562,5.766,148.592
C08022=1211.688,104.760,-49.281,-178.559,5.767,148.591
C08023=1211.684,105.009,-49.300,-178.557,5.768,148.591
C08024=1211.679,105.259,-49.318,-178.555,5.769,148.590
C08025=1211.674,105.508,-49.338,-178.552,5.771,148.590
C08026=1211.670,105.757,-49.356,-178.549,5.771,148.589
C08027=1211.664,106.006,-49.375,-178.547,5.772,148.588
C08028=1211.660,106.255,-49.394,-178.544,5.774,148.588
C08029=1211.655,106.505,-49.413,-178.541,5.774,148.587
C08030=1211.650,106.754,-49.432,-178.539,5.775,148.587
C08031=1211.645,107.022,-49.453,-178.536,5.777,148.586
C08032=1211.639,107.291,-49.473,-178.533,5.777,148.586
C08033=1211.635,107.559,-49.494,-178.531,5.779,148.585
C08034=1211.629,107.828,-49.513,-178.528,5.780,148.584
C08035=1211.625,108.077,-49.533,-178.525,5.781,148.584
C08036=1211.619,108.326,-49.552,-178.523,5.782,148.583
C08037=1211.615,108.575,-49.571,-178.520,5.783,148.583
C08038=1211.610,108.825,-49.590,-178.517,5.784,148.582
C08039=1211.605,109.073,-49.608,-178.515,5.785,148.582
C08040=1211.600,109.323,-49.628,-178.513,5.786,148.581
C08041=1211.596,109.572,-49.647,-178.510,5.787,148.581
C08042=1211.591,109.822,-49.666,-178.507,5.788,148.580
C08043=1211.585,110.071,-49.685,-178.505,5.789,148.580
C08044=1211.581,110.320,-49.704,-178.502,5.791,148.579
C08045=1211.576,110.569,-49.723,-178.499,5.791,148.579
C08046=1211.571,110.818,-49.743,-178.496,5.793,148.578
C08047=1211.567,111.068,-49.762,-178.494,5.794,148.578
C08048=1211.562,111.317,-49.781,-178.492,5.794,148.577
C08049=1211.558,111.566,-49.800,-178.489,5.796,148.577
C08050=1211.552,111.815,-49.819,-178.486,5.796,148.576
C08051=1211.548,112.065,-49.839,-178.484,5.797,148.575
C08052=1211.543,112.313,-49.857,-178.481,5.799,148.575
C08053=1211.538,112.563,-49.877,-178.479,5.800,148.574
C08054=1211.533,112.812,-49.896,-178.476,5.800,148.574
C08055=1211.529,113.061,-49.915,-178.474,5.802,148.573
C08056=1211.524,113.310,-49.935,-178.471,5.803,148.573
C08057=1211.518,113.560,-49.954,-178.468,5.805,148.572
C08058=1211.514,113.810,-49.973,-178.466,5.805,148.572
C08059=1211.509,114.058,-49.992,-178.463,5.806,148.571
C08060=1211.504,114.308,-50.012,-178.460,5.808,148.571
C08061=1211.499,114.557,-50.031,-178.458,5.808,148.570
C08062=1211.495,114.806,-50.050,-178.455,5.810,148.570
C08063=1211.490,115.055,-50.069,-178.453,5.811,148.569
C08064=1211.485,115.304,-50.089,-178.450,5.811,148.569
C08065=1211.480,115.554,-50.109,-178.448,5.813,148.568
C08066=1211.476,115.802,-50.127,-178.445,5.814,148.568
C08067=1211.471,116.052,-50.147,-178.443,5.815,148.567
C08068=1211.466,116.301,-50.166,-178.440,5.816,148.566
C08069=1211.461,116.550,-50.186,-178.438,5.817,148.566
C08070=1211.456,116.800,-50.206,-178.434,5.819,148.565
C08071=1211.451,117.049,-50.224,-178.432,5.820,148.565
C08072=1211.447,117.298,-50.245,-178.430,5.820,148.564
C08073=1211.442,117.546,-50.264,-178.427,5.822,148.564
C08074=1211.437,117.796,-50.284,-178.424,5.823,148.563
C08075=1211.432,118.046,-50.303,-178.422,5.824,148.563
C08076=1211.428,118.294,-50.322,-178.419,5.825,148.562
C08077=1211.423,118.544,-50.342,-178.417,5.826,148.562
C08078=1211.418,118.793,-50.361,-178.414,5.827,148.561
C08079=1211.413,119.042,-50.380,-178.412,5.828,148.561
C08080=1211.408,119.292,-50.400,-178.408,5.830,148.560
C08081=1211.404,119.541,-50.421,-178.406,5.831,148.560
C08082=1211.399,119.789,-50.439,-178.403,5.832,148.559
C08083=1211.394,120.039,-50.459,-178.401,5.833,148.559
C08084=1211.389,120.288,-50.479,-178.398,5.834,148.558
C08085=1211.384,120.537,-50.498,-178.396,5.835,148.558
C08086=1211.380,120.786,-50.518,-178.393,5.836,148.557
C08087=1211.375,121.036,-50.538,-178.390,5.838,148.557
C08088=1211.370,121.285,-50.557,-178.388,5.838,148.556
C08089=1211.365,121.534,-50.577,-178.386,5.839,148.556
C08090=1211.360,121.784,-50.596,-178.383,5.841,148.555
C08091=1211.356,122.033,-50.617,-178.380,5.842,148.555
C08092=1211.351,122.281,-50.636,-178.378,5.844,148.554
C08093=1211.346,122.531,-50.655,-178.375,5.844,148.554
C08094=1211.342,122.780,-50.676,-178.372,5.846,148.553
C08095=1211.337,123.029,-50.695,-178.370,5.847,148.553
C08096=1211.332,123.278,-50.714,-178.368,5.847,148.552
C08097=1211.327,123.528,-50.734,-178.365,5.849,148.552
C08098=1211.323,123.777,-50.755,-178.362,5.850,148.551
C08099=1211.317,124.026,-50.774,-178.359,5.851,148.551
C08100=1211.313,124.275,-50.793,-178.357,5.852,148.550
C08101=1211.308,124.524,-50.814,-178.354,5.854,148.550
C08102=1211.303,124.774,-50.833,-178.352,5.855,148.549
C08103=1211.298,125.022,-50.853,-178.349,5.856,148.549
C08104=1211.294,125.271,-50.873,-178.347,5.857,148.548
C08105=1211.289,125.521,-50.893,-178.344,5.858,148.548
C08106=1211.284,125.770,-50.913,-178.341,5.859,148.547
C08107=1211.279,126.019,-50.932,-178.339,5.860,148.547
C08108=1211.275,126.268,-50.953,-178.336,5.862,148.546
C08109=1211.270,126.517,-50.972,-178.334,5.863,148.546
C08110=1211.265,126.767,-50.992,-178.331,5.864,148.545
C08111=1211.261,127.016,-51.013,-178.329,5.865,148.545
C08112=1211.255,127.265,-51.032,-178.326,5.867,148.544
C08113=1211.251,127.514,-51.052,-178.323,5.868,148.544
C08114=1211.246,127.763,-51.072,-178.321,5.869,148.543
C08115=1211.242,128.012,-51.092,-178.318,5.870,148.543
C08116=1211.236,128.262,-51.112,-178.315,5.872,148.542
C08117=1211.231,128.510,-51.132,-178.313,5.872,148.542
C08118=1211.226,128.760,-51.152,-178.311,5.873,148.541
C08119=1211.222,129.009,-51.173,-178.308,5.875,148.541
C08120=1211.217,129.258,-51.192,-178.305,5.876,148.540
C08121=1211.213,129.507,-51.213,-178.303,5.878,148.540
C08122=1211.208,129.757,-51.232,-178.300,5.878,148.539
C08123=1211.203,130.005,-51.252,-178.297,5.880,148.539
C08124=1211.199,130.254,-51.273,-178.295,5.881,148.538
C08125=1211.193,130.504,-51.293,-178.292,5.882,148.538
C08126=1211.189,130.753,-51.313,-178.290,5.883,148.537
C08127=1211.184,131.003,-51.333,-178.287,5.885,148.537
C08128=1211.180,131.251,-51.353,-178.285,5.886,148.536
C08129=1211.175,131.500,-51.374,-178.281,5.887,148.536
C08130=1211.170,131.749,-51.393,-178.279,5.888,148.535
C08131=1211.165,131.999,-51.414,-178.277,5.890,148.535
C08132=1211.160,132.247,-51.434,-178.274,5.890,148.534
C08133=1211.155,132.497,-51.454,-178.271,5.892,148.534
C08134=1211.151,132.746,-51.474,-178.269,5.893,148.533
C08135=1211.145,133.015,-51.496,-178.266,5.895,148.533
C08136=1211.141,133.283,-51.518,-178.263,5.896,148.532
C08137=1211.135,133.552,-51.539,-178.261,5.897,148.532
C08138=1211.130,133.820,-51.562,-178.258,5.899,148.531
C08139=1211.125,134.069,-51.582,-178.255,5.899,148.531
C08140=1211.120,134.319,-51.602,-178.252,5.901,148.530
C08141=1211.116,134.568,-51.622,-178.250,5.902,148.530
C08142=1211.111,134.817,-51.643,-178.247,5.903,148.529
C08143=1211.106,135.066,-51.664,-178.245,5.904,148.529
C08144=1211.102,135.316,-51.683,-178.242,5.906,148.528
C08145=1211.097,135.564,-51.704,-178.240,5.907,148.528
C08146=1211.092,135.814,-51.725,-178.237,5.908,148.527
C08147=1211.088,136.063,-51.745,-178.234,5.910,148.527
C08148=1211.083,136.312,-51.765,-178.232,5.911,148.526
C08149=1211.078,136.562,-51.786,-178.229,5.913,148.526
C08150=1211.073,136.810,-51.806,-178.226,5.913,148.525
C08151=1211.069,137.059,-51.826,-178.224,5.915,148.525
C08152=1211.064,137.309,-51.847,-178.221,5.916,148.524
C08153=1211.059,137.558,-51.868,-178.218,5.917,148.524
C08154=1211.055,137.807,-51.888,-178.216,5.918,148.524
C08155=1211.049,138.056,-51.908,-178.213,5.920,148.523
C08156=1211.044,138.305,-51.928,-178.211,5.921,148.523
C08157=1211.040,138.554,-51.949,-178.208,5.923,148.522
C08158=1211.035,138.803,-51.970,-178.206,5.923,148.522
C08159=1211.030,139.052,-51.990,-178.203,5.925,148.521
C08160=1211.026,139.301,-52.010,-178.200,5.926,148.521
C08161=1211.021,139.550,-52.031,-178.198,5.927,148.520
C08162=1211.016,139.799,-52.052,-178.196,5.928,148.520
C08163=1211.011,140.048,-52.073,-178.193,5.930,148.519
C08164=1211.007,140.297,-52.093,-178.190,5.931,148.519
C08165=1211.003,140.547,-52.114,-178.188,5.933,148.518
C08166=1210.998,140.796,-52.135,-178.185,5.934,148.518
C08167=1210.993,141.045,-52.155,-178.182,5.935,148.517
C08168=1210.988,141.294,-52.176,-178.180,5.937,148.517
C08169=1210.984,141.543,-52.196,-178.177,5.937,148.516
C08170=1210.978,141.793,-52.217,-178.175,5.939,148.516
C08171=1210.974,142.042,-52.238,-178.172,5.940,148.515
C08172=1210.969,142.291,-52.259,-178.169,5.942,148.515
C08173=1210.964,142.540,-52.279,-178.167,5.943,148.515
C08174=1210.960,142.789,-52.299,-178.164,5.944,148.514
C08175=1210.955,143.038,-52.320,-178.161,5.946,148.514
C08176=1210.950,143.287,-52.341,-178.159,5.947,148.513
C08177=1210.945,143.536,-52.362,-178.156,5.948,148.513
C08178=1210.941,143.785,-52.382,-178.154,5.949,148.512
C08179=1210.936,144.034,-52.404,-178.151,5.951,148.512
C08180=1210.931,144.283,-52.424,-178.149,5.952,148.511
C08181=1210.926,144.532,-52.445,-178.146,5.954,148.511
C08182=1210.922,144.782,-52.467,-178.144,5.954,148.510
C08183=1210.917,145.031,-52.487,-178.141,5.956,148.510
C08184=1210.912,145.280,-52.508,-178.138,5.958,148.509
C08185=1210.908,145.529,-52.528,-178.136,5.959,148.509
C08186=1210.903,145.778,-52.550,-178.133,5.960,148.508
C08187=1210.898,146.027,-52.570,-178.131,5.961,148.508
C08188=1210.893,146.276,-52.591,-178.128,5.963,148.508
C08189=1210.889,146.525,-52.612,-178.125,5.964,148.507
C08190=1210.884,146.773,-52.633,-178.123,5.965,148.507
C08191=1210.879,147.023,-52.655,-178.120,5.967,148.506
C08192=1210.875,147.272,-52.675,-178.117,5.968,148.506
C08193=1210.870,147.522,-52.696,-178.115,5.970,148.505
C08194=1210.865,147.770,-52.717,-178.113,5.971,148.505
C08195=1210.860,148.019,-52.738,-178.109,5.972,148.504
C08196=1210.855,148.269,-52.759,-178.107,5.974,148.504
C08197=1210.851,148.517,-52.779,-178.105,5.975,148.503
C08198=1210.846,148.767,-52.801,-178.102,5.977,148.503
C08199=1210.841,149.016,-52.822,-178.099,5.977,148.502
C08200=1210.837,149.265,-52.843,-178.097,5.979,148.502
C08201=1210.832,149.514,-52.864,-178.094,5.981,148.502
C08202=1210.827,149.763,-52.885,-178.091,5.981,148.501
C08203=1210.823,150.013,-52.906,-178.089,5.983,148.501
C08204=1210.818,150.261,-52.928,-178.087,5.984,148.500
C08205=1210.813,150.510,-52.949,-178.084,5.986,148.500
C08206=1210.809,150.759,-52.970,-178.081,5.987,148.499
C08207=1210.804,151.008,-52.991,-178.079,5.988,148.499
C08208=1210.798,151.257,-53.012,-178.076,5.990,148.498
C08209=1210.795,151.506,-53.033,-178.073,5.991,148.498
C08210=1210.790,151.756,-53.054,-178.071,5.993,148.498
C08211=1210.785,152.004,-53.076,-178.068,5.994,148.497
C08212=1210.780,152.253,-53.097,-178.066,5.995,148.497
C08213=1210.776,152.503,-53.118,-178.063,5.997,148.496
C08214=1210.771,152.752,-53.139,-178.060,5.999,148.496
C08215=1210.766,153.001,-53.160,-178.058,5.999,148.495
C08216=1210.761,153.250,-53.182,-178.055,6.001,148.495
C08217=1210.756,153.499,-53.202,-178.053,6.002,148.494
C08218=1210.752,153.748,-53.224,-178.050,6.004,148.494
C08219=1210.747,153.997,-53.246,-178.047,6.005,148.493
C08220=1210.742,154.246,-53.267,-178.045,6.006,148.493
C08221=1210.738,154.495,-53.289,-178.042,6.008,148.493
C08222=1210.733,154.744,-53.309,-178.039,6.010,148.492
C08223=1210.729,154.993,-53.331,-178.037,6.011,148.492
C08224=1210.723,155.242,-53.352,-178.034,6.012,148.491
C08225=1210.719,155.491,-53.374,-178.032,6.013,148.491
C08226=1210.714,155.741,-53.395,-178.029,6.015,148.490
C08227=1210.710,155.989,-53.416,-178.026,6.017,148.490
C08228=1210.705,156.238,-53.438,-178.024,6.018,148.490
C08229=1210.700,156.488,-53.459,-178.022,6.019,148.489
C08230=1210.695,156.736,-53.481,-178.018,6.021,148.489
C08231=1210.691,156.985,-53.503,-178.016,6.022,148.488
C08232=1210.686,157.235,-53.524,-178.014,6.024,148.488
C08233=1210.681,157.483,-53.546,-178.011,6.025,148.487
C08234=1210.676,157.732,-53.567,-178.008,6.026,148.487
C08235=1210.672,157.982,-53.588,-178.006,6.028,148.486
C08236=1210.668,158.230,-53.610,-178.003,6.030,148.486
C08237=1210.663,158.479,-53.631,-178.001,6.031,148.486
C08238=1210.658,158.729,-53.653,-177.998,6.032,148.485
C08239=1210.653,158.998,-53.677,-177.995,6.034,148.485
C08240=1210.648,159.267,-53.700,-177.992,6.035,148.484
C08241=1210.643,159.536,-53.723,-177.990,6.036,148.484
C08242=1210.638,159.805,-53.746,-177.987,6.038,148.483
C08243=1210.633,160.054,-53.767,-177.984,6.040,148.483
C08244=1210.628,160.302,-53.789,-177.981,6.041,148.482
C08245=1210.624,160.552,-53.811,-177.979,6.042,148.482
C08246=1210.619,160.800,-53.833,-177.977,6.044,148.482
C08247=1210.614,161.050,-53.854,-177.973,6.046,148.481
C08248=1210.610,161.299,-53.876,-177.971,6.047,148.481
C08249=1210.605,161.548,-53.897,-177.969,6.048,148.480
C08250=1210.601,161.797,-53.919,-177.966,6.050,148.480
C08251=1210.596,162.046,-53.941,-177.963,6.051,148.479
C08252=1210.591,162.294,-53.963,-177.961,6.053,148.479
C08253=1210.587,162.544,-53.985,-177.958,6.054,148.479
C08254=1210.581,162.793,-54.006,-177.956,6.055,148.478
C08255=1210.577,163.042,-54.028,-177.953,6.057,148.478
C08256=1210.572,163.291,-54.050,-177.950,6.059,148.477
C08257=1210.567,163.540,-54.071,-177.948,6.061,148.477
C08258=1210.563,163.789,-54.093,-177.945,6.062,148.476
C08259=1210.558,164.038,-54.115,-177.943,6.063,148.476
C08260=1210.554,164.287,-54.137,-177.940,6.065,148.476
C08261=1210.548,164.536,-54.159,-177.937,6.066,148.475
C08262=1210.544,164.785,-54.181,-177.935,6.068,148.475
C08263=1210.539,165.034,-54.203,-177.932,6.069,148.474
C08264=1210.534,165.282,-54.225,-177.930,6.070,148.474
C08265=1210.530,165.532,-54.247,-177.927,6.072,148.473
C08266=1210.525,165.780,-54.268,-177.924,6.074,148.473
C08267=1210.521,166.030,-54.291,-177.922,6.075,148.473
C08268=1210.516,166.278,-54.312,-177.919,6.076,148.472
C08269=1210.512,166.528,-54.334,-177.917,6.078,148.472
C08270=1210.507,166.776,-54.356,-177.914,6.080,148.471
C08271=1210.502,167.026,-54.379,-177.912,6.081,148.471
C08272=1210.497,167.275,-54.400,-177.909,6.082,148.471
C08273=1210.493,167.524,-54.422,-177.906,6.084,148.470
C08274=1210.488,167.773,-54.444,-177.904,6.085,148.470
C08275=1210.484,168.022,-54.466,-177.901,6.087,148.469
C08276=1210.479,168.271,-54.488,-177.898,6.089,148.469
C08277=1210.474,168.520,-54.510,-177.896,6.090,148.469
C08278=1210.469,168.768,-54.533,-177.894,6.091,148.468
C08279=1210.465,169.018,-54.555,-177.891,6.093,148.468
C08280=1210.460,169.266,-54.577,-177.888,6.095,148.467
C08281=1210.456,169.516,-54.599,-177.885,6.096,148.467
C08282=1210.450,169.765,-54.621,-177.883,6.097,148.466
C08283=1210.446,170.014,-54.643,-177.880,6.099,148.466
C08284=1210.441,170.262,-54.665,-177.878,6.101,148.466
C08285=1210.437,170.511,-54.687,-177.875,6.102,148.465
C08286=1210.431,170.760,-54.710,-177.872,6.104,148.465
C08287=1210.427,171.010,-54.732,-177.870,6.105,148.464
C08288=1210.423,171.259,-54.754,-177.867,6.107,148.464
C08289=1210.418,171.507,-54.776,-177.865,6.108,148.464
C08290=1210.413,171.757,-54.799,-177.862,6.110,148.463
C08291=1210.409,172.005,-54.820,-177.859,6.111,148.463
C08292=1210.404,172.255,-54.842,-177.857,6.113,148.462
C08293=1210.399,172.503,-54.865,-177.854,6.114,148.462
C08294=1210.395,172.752,-54.888,-177.852,6.116,148.462
C08295=1210.390,173.002,-54.910,-177.849,6.118,148.461
C08296=1210.385,173.250,-54.933,-177.846,6.120,148.461
C08297=1210.381,173.499,-54.955,-177.844,6.120,148.460
C08298=1210.376,173.748,-54.976,-177.841,6.122,148.460
C08299=1210.371,173.997,-55.000,-177.839,6.124,148.459
C08300=1210.367,174.246,-55.022,-177.836,6.126,148.459
C08301=1210.362,174.495,-55.043,-177.834,6.127,148.459
C08302=1210.357,174.744,-55.067,-177.831,6.129,148.458
C08303=1210.353,174.993,-55.088,-177.828,6.130,148.458
C08304=1210.349,175.241,-55.111,-177.825,6.132,148.457
C08305=1210.344,175.491,-55.134,-177.823,6.133,148.457
C08306=1210.339,175.740,-55.156,-177.821,6.135,148.457
C08307=1210.334,175.989,-55.179,-177.818,6.136,148.456
C08308=1210.330,176.238,-55.201,-177.815,6.138,148.456
C08309=1210.325,176.486,-55.223,-177.813,6.140,148.456
C08310=1210.320,176.736,-55.246,-177.810,6.141,148.455
C08311=1210.316,176.984,-55.269,-177.807,6.143,148.455
C08312=1210.311,177.233,-55.291,-177.805,6.144,148.454
C08313=1210.307,177.482,-55.314,-177.802,6.146,148.454
C08314=1210.302,177.732,-55.336,-177.800,6.147,148.454
C08315=1210.297,177.980,-55.359,-177.797,6.149,148.453
C08316=1210.293,178.229,-55.381,-177.795,6.151,148.453
C08317=1210.288,178.478,-55.404,-177.792,6.153,148.452
C08318=1210.283,178.727,-55.426,-177.789,6.154,148.452
C08319=1210.279,178.976,-55.449,-177.787,6.155,148.452
C08320=1210.274,179.225,-55.471,-177.784,6.157,148.451
C08321=1210.269,179.473,-55.494,-177.781,6.159,148.451
C08322=1210.265,179.723,-55.516,-177.779,6.161,148.450
C08323=1210.260,179.972,-55.540,-177.776,6.162,148.450
C08324=1210.256,180.221,-55.562,-177.774,6.163,148.450
C08325=1210.250,180.469,-55.585,-177.771,6.165,148.449
C08326=1210.246,180.718,-55.608,-177.769,6.167,148.449
C08327=1210.242,180.967,-55.631,-177.765,6.168,148.448
C08328=1210.237,181.216,-55.653,-177.763,6.170,148.448
C08329=1210.232,181.465,-55.676,-177.761,6.171,148.448
C08330=1210.228,181.714,-55.699,-177.758,6.173,148.447
C08331=1210.223,181.963,-55.721,-177.755,6.175,148.447
C08332=1210.218,182.212,-55.744,-177.753,6.177,148.447
C08333=1210.214,182.460,-55.767,-177.750,6.179,148.446
C08334=1210.209,182.710,-55.790,-177.748,6.180,148.446
C08335=1210.205,182.959,-55.812,-177.745,6.181,148.446
C08336=1210.200,183.207,-55.835,-177.743,6.183,148.445
C08337=1210.195,183.456,-55.859,-177.740,6.185,148.445
C08338=1210.191,183.705,-55.881,-177.737,6.186,148.444
C08339=1210.186,183.954,-55.904,-177.734,6.188,148.444
C08340=1210.181,184.203,-55.928,-177.732,6.189,148.444
C08341=1210.177,184.451,-55.950,-177.730,6.191,148.443
C08342=1210.172,184.701,-55.973,-177.727,6.193,148.443
C08343=1210.167,184.971,-55.997,-177.724,6.195,148.442
C08344=1210.162,185.240,-56.023,-177.721,6.196,148.442
C08345=1210.157,185.510,-56.048,-177.718,6.198,148.442
C08346=1210.152,185.779,-56.072,-177.716,6.200,148.441
C08347=1210.148,186.028,-56.096,-177.713,6.202,148.441
C08348=1210.143,186.278,-56.118,-177.710,6.203,148.440
C08349=1210.139,186.526,-56.141,-177.708,6.205,148.440
C08350=1210.134,186.775,-56.164,-177.705,6.207,148.440
C08351=1210.129,187.024,-56.187,-177.703,6.208,148.439
C08352=1210.125,187.272,-56.210,-177.700,6.210,148.439
C08353=1210.120,187.521,-56.234,-177.697,6.211,148.438
C08354=1210.115,187.771,-56.257,-177.695,6.213,148.438
C08355=1210.111,188.020,-56.280,-177.692,6.215,148.438
C08356=1210.107,188.268,-56.303,-177.689,6.217,148.437
C08357=1210.102,188.517,-56.326,-177.687,6.219,148.437
C08358=1210.097,188.766,-56.349,-177.685,6.220,148.437
C08359=1210.092,189.015,-56.373,-177.682,6.222,148.436
C08360=1210.087,189.264,-56.396,-177.679,6.223,148.436
C08361=1210.083,189.512,-56.419,-177.677,6.225,148.436
C08362=1210.079,189.761,-56.442,-177.674,6.227,148.435
C08363=1210.074,190.010,-56.466,-177.671,6.229,148.435
C08364=1210.069,190.260,-56.489,-177.669,6.231,148.435
C08365=1210.064,190.509,-56.512,-177.667,6.232,148.434
C08366=1210.060,190.757,-56.535,-177.664,6.233,148.434
C08367=1210.055,191.006,-56.558,-177.661,6.235,148.433
C08368=1210.050,191.255,-56.581,-177.659,6.237,148.433
C08369=1210.046,191.504,-56.605,-177.656,6.239,148.433
C08370=1210.041,191.753,-56.628,-177.653,6.241,148.432
C08371=1210.036,192.002,-56.651,-177.651,6.243,148.432
C08372=1210.032,192.250,-56.674,-177.647,6.244,148.432
C08373=1210.028,192.499,-56.698,-177.645,6.245,148.431
C08374=1210.023,192.748,-56.722,-177.643,6.247,148.431
C08375=1210.019,192.997,-56.745,-177.640,6.249,148.430
C08376=1210.014,193.246,-56.768,-177.637,6.251,148.430
C08377=1210.009,193.495,-56.792,-177.635,6.252,148.430
C08378=1210.005,193.744,-56.815,-177.632,6.254,148.429
C08379=1210.000,193.993,-56.838,-177.629,6.256,148.429
C08380=1209.995,194.241,-56.863,-177.627,6.258,148.429
C08381=1209.991,194.491,-56.886,-177.625,6.259,148.428
C08382=1209.987,194.739,-56.909,-177.622,6.261,148.428
C08383=1209.981,194.988,-56.932,-177.619,6.263,148.428
C08384=1209.977,195.236,-56.956,-177.617,6.264,148.427
C08385=1209.972,195.485,-56.979,-177.614,6.266,148.427
C08386=1209.968,195.734,-57.002,-177.612,6.268,148.427
C08387=1209.963,195.983,-57.026,-177.609,6.270,148.426
C08388=1209.959,196.231,-57.050,-177.606,6.272,148.426
C08389=1209.954,196.481,-57.073,-177.604,6.273,148.426
C08390=1209.949,196.730,-57.097,-177.601,6.275,148.425
C08391=1209.945,196.978,-57.121,-177.598,6.277,148.425
C08392=1209.941,197.228,-57.144,-177.596,6.278,148.425
C08393=1209.936,197.477,-57.168,-177.594,6.280,148.424
C08394=1209.932,197.725,-57.192,-177.591,6.282,148.424
C08395=1209.927,197.974,-57.215,-177.588,6.284,148.423
C08396=1209.922,198.223,-57.239,-177.586,6.285,148.423
C08397=1209.918,198.472,-57.263,-177.583,6.287,148.423
C08398=1209.913,198.721,-57.286,-177.580,6.289,148.422
C08399=1209.908,198.969,-57.311,-177.578,6.291,148.422
C08400=1209.903,199.218,-57.334,-177.575,6.293,148.422
C08401=1209.899,199.467,-57.358,-177.572,6.295,148.421
C08402=1209.894,199.716,-57.381,-177.570,6.296,148.421
C08403=1209.889,199.965,-57.405,-177.567,6.298,148.421
C08404=1209.885,200.213,-57.429,-177.565,6.299,148.420
C08405=1209.880,200.462,-57.452,-177.562,6.301,148.420
C08406=1209.876,200.711,-57.476,-177.560,6.303,148.420
C08407=1209.871,200.960,-57.500,-177.557,6.305,148.419
C08408=1209.867,201.208,-57.524,-177.554,6.307,148.419
C08409=1209.863,201.458,-57.547,-177.552,6.308,148.419
C08410=1209.858,201.707,-57.572,-177.549,6.310,148.418
C08411=1209.853,201.956,-57.596,-177.546,6.312,148.418
C08412=1209.849,202.204,-57.620,-177.544,6.314,148.418
C08413=1209.844,202.452,-57.644,-177.541,6.316,148.417
C08414=1209.839,202.702,-57.667,-177.538,6.318,148.417
C08415=1209.835,202.950,-57.691,-177.536,6.319,148.417
C08416=1209.830,203.199,-57.715,-177.533,6.321,148.416
C08417=1209.826,203.448,-57.739,-177.531,6.323,148.416
C08418=1209.821,203.697,-57.764,-177.528,6.325,148.416
C08419=1209.817,203.946,-57.787,-177.526,6.327,148.415
C08420=1209.812,204.194,-57.811,-177.523,6.329,148.415
C08421=1209.807,204.443,-57.836,-177.520,6.331,148.415
C08422=1209.803,204.692,-57.859,-177.518,6.333,148.414
C08423=1209.798,204.940,-57.883,-177.516,6.334,148.414
C08424=1209.794,205.190,-57.908,-177.513,6.335,148.414
C08425=1209.790,205.439,-57.931,-177.510,6.337,148.413
C08426=1209.784,205.687,-57.956,-177.508,6.339,148.413
C08427=1209.780,205.936,-57.980,-177.505,6.341,148.413
C08428=1209.775,206.185,-58.003,-177.502,6.343,148.412
C08429=1209.771,206.434,-58.028,-177.500,6.345,148.412
C08430=1209.766,206.683,-58.052,-177.497,6.346,148.412
C08431=1209.762,206.931,-58.076,-177.495,6.348,148.411
C08432=1209.757,207.180,-58.100,-177.492,6.350,148.411
C08433=1209.752,207.429,-58.124,-177.489,6.352,148.411
C08434=1209.748,207.678,-58.149,-177.487,6.354,148.410
C08435=1209.744,207.926,-58.173,-177.484,6.356,148.410
C08436=1209.739,208.175,-58.197,-177.482,6.358,148.410
C08437=1209.734,208.424,-58.221,-177.479,6.360,148.410
C08438=1209.730,208.672,-58.245,-177.477,6.361,148.409
C08439=1209.725,208.922,-58.270,-177.474,6.363,148.409
C08440=1209.721,209.170,-58.294,-177.471,6.365,148.409
C08441=1209.716,209.419,-58.319,-177.469,6.367,148.408
C08442=1209.711,209.667,-58.343,-177.466,6.369,148.408
C08443=1209.708,209.917,-58.367,-177.463,6.371,148.408
C08444=1209.702,210.165,-58.392,-177.461,6.372,148.407
C08445=1209.698,210.414,-58.415,-177.458,6.374,148.407
C08446=1209.693,210.663,-58.439,-177.455,6.376,148.406
C08447=1209.689,210.934,-58.466,-177.453,6.378,148.406
C08448=1209.684,211.204,-58.493,-177.450,6.381,148.406
C08449=1209.679,211.474,-58.520,-177.447,6.382,148.406
C08450=1209.673,211.745,-58.546,-177.444,6.384,148.405
C08451=1209.669,211.994,-58.570,-177.442,6.386,148.405
C08452=1209.664,212.243,-58.595,-177.439,6.388,148.405
C08453=1209.660,212.491,-58.619,-177.436,6.390,148.404
C08454=1209.655,212.740,-58.644,-177.434,6.392,148.404
C08455=1209.651,212.989,-58.668,-177.431,6.393,148.404
C08456=1209.646,213.237,-58.693,-177.429,6.396,148.403
C08457=1209.642,213.485,-58.717,-177.426,6.397,148.403
C08458=1209.638,213.734,-58.742,-177.424,6.399,148.403
C08459=1209.633,213.983,-58.767,-177.421,6.401,148.402
C08460=1209.628,214.232,-58.791,-177.418,6.403,148.402
C08461=1209.624,214.481,-58.816,-177.416,6.405,148.402
C08462=1209.619,214.730,-58.840,-177.413,6.407,148.401
C08463=1209.614,214.978,-58.864,-177.410,6.408,148.401
C08464=1209.610,215.228,-58.889,-177.408,6.410,148.401
C08465=1209.605,215.476,-58.914,-177.405,6.413,148.401
C08466=1209.600,215.724,-58.939,-177.402,6.415,148.400
C08467=1209.597,215.973,-58.963,-177.400,6.417,148.400
C08468=1209.592,216.222,-58.988,-177.397,6.419,148.400
C08469=1209.588,216.471,-59.012,-177.395,6.421,148.399
C08470=1209.583,216.720,-59.037,-177.392,6.422,148.399
C08471=1209.577,216.968,-59.062,-177.389,6.424,148.399
C08472=1209.574,217.217,-59.087,-177.387,6.426,148.398
C08473=1209.569,217.466,-59.112,-177.384,6.428,148.398
C08474=1209.564,217.714,-59.136,-177.382,6.430,148.398
C08475=1209.560,217.964,-59.161,-177.379,6.432,148.398
C08476=1209.555,218.212,-59.186,-177.377,6.434,148.397
C08477=1209.551,218.461,-59.211,-177.374,6.436,148.397
C08478=1209.546,218.709,-59.235,-177.371,6.438,148.397
C08479=1209.542,218.958,-59.261,-177.369,6.439,148.396
C08480=1209.538,219.207,-59.285,-177.366,6.442,148.396
C08481=1209.532,219.455,-59.310,-177.364,6.443,148.396
C08482=1209.528,219.704,-59.335,-177.361,6.445,148.395
C08483=1209.524,219.953,-59.360,-177.359,6.447,148.395
C08484=1209.519,220.202,-59.385,-177.356,6.449,148.395
C08485=1209.514,220.450,-59.410,-177.353,6.451,148.394
C08486=1209.511,220.699,-59.434,-177.351,6.453,148.394
C08487=1209.506,220.948,-59.459,-177.348,6.456,148.394
C08488=1209.501,221.197,-59.485,-177.345,6.457,148.394
C08489=1209.497,221.445,-59.509,-177.343,6.459,148.393
C08490=1209.493,221.694,-59.535,-177.340,6.461,148.393
C08491=1209.488,221.943,-59.559,-177.337,6.463,148.393
C08492=1209.482,222.191,-59.584,-177.335,6.465,148.393
C08493=1209.479,222.440,-59.609,-177.333,6.467,148.392
C08494=1209.474,222.689,-59.634,-177.330,6.469,148.392
C08495=1209.470,222.937,-59.660,-177.327,6.471,148.392
C08496=1209.464,223.186,-59.684,-177.325,6.472,148.391
C08497=1209.461,223.435,-59.709,-177.322,6.474,148.391
C08498=1209.456,223.683,-59.734,-177.320,6.476,148.391
C08499=1209.452,223.932,-59.760,-177.317,6.478,148.391
C08500=1209.446,224.181,-59.785,-177.315,6.480,148.390
C08501=1209.442,224.430,-59.810,-177.312,6.482,148.390
C08502=1209.438,224.678,-59.834,-177.309,6.485,148.390
C08503=1209.434,224.927,-59.860,-177.307,6.487,148.390
C08504=1209.429,225.176,-59.886,-177.304,6.489,148.389
C08505=1209.424,225.424,-59.911,-177.301,6.491,148.389
C08506=1209.420,225.673,-59.936,-177.299,6.492,148.389
C08507=1209.415,225.922,-59.961,-177.296,6.494,148.388
C08508=1209.411,226.171,-59.987,-177.294,6.496,148.388
C08509=1209.407,226.419,-60.011,-177.291,6.498,148.388
C08510=1209.402,226.668,-60.036,-177.289,6.500,148.387
C08511=1209.397,226.916,-60.062,-177.286,6.502,148.387
C08512=1209.393,227.165,-60.088,-177.283,6.504,148.387
C08513=1209.388,227.414,-60.113,-177.281,6.506,148.387
C08514=1209.384,227.662,-60.138,-177.278,6.509,148.386
C08515=1209.379,227.911,-60.164,-177.275,6.510,148.386
C08516=1209.374,228.160,-60.188,-177.273,6.512,148.386
C08517=1209.370,228.409,-60.214,-177.271,6.515,148.386
C08518=1209.365,228.657,-60.240,-177.268,6.516,148.385
C08519=1209.361,228.906,-60.265,-177.265,6.518,148.385
C08520=1209.357,229.155,-60.290,-177.263,6.520,148.385
C08521=1209.352,229.403,-60.316,-177.260,6.522,148.384
C08522=1209.348,229.652,-60.341,-177.258,6.524,148.384
C08523=1209.344,229.901,-60.367,-177.255,6.526,148.384
C08524=1209.339,230.149,-60.392,-177.253,6.528,148.384
C08525=1209.335,230.398,-60.417,-177.249,6.530,148.383
C08526=1209.330,230.646,-60.442,-177.247,6.533,148.383
C08527=1209.326,230.895,-60.468,-177.245,6.534,148.383
C08528=1209.321,231.144,-60.494,-177.242,6.536,148.383
C08529=1209.317,231.392,-60.519,-177.239,6.538,148.382
C08530=1209.312,231.641,-60.545,-177.237,6.540,148.382
C08531=1209.307,231.890,-60.571,-177.235,6.542,148.382
C08532=1209.302,232.139,-60.596,-177.232,6.544,148.381
C08533=1209.298,232.387,-60.622,-177.229,6.546,148.381
C08534=1209.294,232.636,-60.648,-177.227,6.549,148.381
C08535=1209.289,232.884,-60.673,-177.224,6.551,148.381
C08536=1209.285,233.133,-60.699,-177.221,6.553,148.380
C08537=1209.280,233.382,-60.725,-177.219,6.555,148.380
C08538=1209.276,233.630,-60.750,-177.217,6.557,148.380
C08539=1209.271,233.879,-60.776,-177.214,6.558,148.380
C08540=1209.267,234.128,-60.801,-177.211,6.560,148.379
C08541=1209.263,234.376,-60.827,-177.209,6.562,148.379
C08542=1209.258,234.624,-60.853,-177.206,6.565,148.379
C08543=1209.253,234.874,-60.879,-177.203,6.567,148.379
C08544=1209.249,235.122,-60.905,-177.201,6.569,148.379
C08545=1209.244,235.370,-60.930,-177.199,6.571,148.378
C08546=1209.240,235.619,-60.956,-177.196,6.573,148.378
C08547=1209.236,235.868,-60.982,-177.193,6.575,148.378
C08548=1209.231,236.117,-61.007,-177.191,6.577,148.378
C08549=1209.227,236.365,-61.033,-177.189,6.579,148.377
C08550=1209.222,236.614,-61.059,-177.185,6.581,148.377
C08551=1209.217,236.885,-61.088,-177.183,6.583,148.377
C08552=1209.212,237.157,-61.115,-177.181,6.585,148.377
C08553=1209.207,237.428,-61.143,-177.177,6.588,148.376
C08554=1209.203,237.700,-61.172,-177.175,6.590,148.376
C08555=1209.198,237.948,-61.198,-177.172,6.593,148.376
C08556=1209.193,238.197,-61.224,-177.169,6.595,148.375
C08557=1209.189,238.446,-61.250,-177.167,6.597,148.375
C08558=1209.185,238.694,-61.276,-177.164,6.599,148.375
C08559=1209.180,238.942,-61.302,-177.162,6.600,148.375
C08560=1209.175,239.191,-61.328,-177.159,6.603,148.374
C08561=1209.171,239.440,-61.354,-177.157,6.604,148.374
C08562=1209.167,239.689,-61.379,-177.154,6.607,148.374
C08563=1209.163,239.937,-61.406,-177.151,6.609,148.374
C08564=1209.157,240.185,-61.432,-177.149,6.611,148.373
C08565=1209.153,240.434,-61.458,-177.146,6.613,148.373
C08566=1209.149,240.683,-61.483,-177.144,6.615,148.373
C08567=1209.144,240.932,-61.510,-177.141,6.617,148.373
C08568=1209.140,241.180,-61.536,-177.138,6.620,148.372
C08569=1209.136,241.429,-61.562,-177.136,6.622,148.372
C08570=1209.130,241.677,-61.589,-177.133,6.624,148.372
C08571=1209.126,241.926,-61.614,-177.131,6.626,148.372
C08572=1209.122,242.175,-61.640,-177.129,6.628,148.372
C08573=1209.117,242.423,-61.667,-177.126,6.630,148.371
C08574=1209.113,242.672,-61.693,-177.123,6.632,148.371
C08575=1209.109,242.921,-61.719,-177.121,6.634,148.371
C08576=1209.104,243.169,-61.746,-177.118,6.636,148.371
C08577=1209.099,243.417,-61.771,-177.116,6.638,148.370
C08578=1209.095,243.666,-61.798,-177.113,6.640,148.370
C08579=1209.091,243.915,-61.824,-177.111,6.642,148.370
C08580=1209.087,244.163,-61.850,-177.108,6.645,148.370
C08581=1209.082,244.412,-61.877,-177.105,6.647,148.370
C08582=1209.078,244.660,-61.903,-177.103,6.649,148.369
C08583=1209.073,244.909,-61.930,-177.101,6.651,148.369
C08584=1209.069,245.158,-61.955,-177.098,6.653,148.369
C08585=1209.065,245.406,-61.982,-177.095,6.656,148.369
C08586=1209.059,245.655,-62.008,-177.093,6.658,148.368
C08587=1209.055,245.903,-62.034,-177.090,6.660,148.368
C08588=1209.050,246.151,-62.061,-177.087,6.662,148.368
C08589=1209.046,246.400,-62.087,-177.085,6.664,148.368
C08590=1209.042,246.649,-62.114,-177.082,6.666,148.367
C08591=1209.037,246.897,-62.140,-177.080,6.669,148.367
C08592=1209.033,247.146,-62.167,-177.077,6.670,148.367
C08593=1209.028,247.395,-62.193,-177.075,6.672,148.367
C08594=1209.024,247.643,-62.220,-177.073,6.675,148.367
C08595=1209.020,247.891,-62.246,-177.069,6.677,148.366
C08596=1209.015,248.140,-62.273,-177.067,6.679,148.366
C08597=1209.011,248.389,-62.299,-177.065,6.681,148.366
C08598=1209.006,248.638,-62.325,-177.062,6.683,148.366
C08599=1209.001,248.886,-62.352,-177.059,6.686,148.366
C08600=1208.997,249.134,-62.379,-177.057,6.688,148.365
C08601=1208.993,249.383,-62.406,-177.055,6.690,148.365
C08602=1208.989,249.632,-62.432,-177.052,6.692,148.365
C08603=1208.984,249.880,-62.459,-177.049,6.694,148.365
C08604=1208.980,250.128,-62.485,-177.047,6.697,148.365
C08605=1208.975,250.377,-62.512,-177.044,6.699,148.364
C08606=1208.970,250.626,-62.539,-177.042,6.701,148.364
C08607=1208.967,250.874,-62.565,-177.039,6.703,148.364
C08608=1208.962,251.123,-62.592,-177.036,6.706,148.364
C08609=1208.958,251.371,-62.618,-177.034,6.708,148.363
C08610=1208.953,251.620,-62.645,-177.031,6.709,148.363
C08611=1208.948,251.868,-62.672,-177.029,6.712,148.363
C08612=1208.944,252.117,-62.699,-177.026,6.714,148.363
C08613=1208.940,252.365,-62.726,-177.024,6.717,148.363
C08614=1208.935,252.614,-62.752,-177.021,6.718,148.362
C08615=1208.931,252.862,-62.778,-177.019,6.721,148.362
C08616=1208.926,253.111,-62.805,-177.016,6.722,148.362
C08617=1208.922,253.359,-62.833,-177.013,6.725,148.362
C08618=1208.918,253.608,-62.859,-177.011,6.727,148.362
C08619=1208.913,253.856,-62.886,-177.008,6.729,148.361
C08620=1208.908,254.105,-62.913,-177.006,6.731,148.361
C08621=1208.904,254.353,-62.940,-177.003,6.734,148.361
C08622=1208.900,254.601,-62.967,-177.001,6.736,148.361
C08623=1208.895,254.851,-62.993,-176.998,6.738,148.361
C08624=1208.891,255.100,-63.020,-176.996,6.740,148.361
C08625=1208.886,255.348,-63.047,-176.993,6.743,148.360
C08626=1208.882,255.596,-63.074,-176.990,6.745,148.360
C08627=1208.877,255.845,-63.101,-176.988,6.747,148.360
C08628=1208.873,256.093,-63.128,-176.985,6.750,148.360
C08629=1208.868,256.342,-63.155,-176.983,6.752,148.359
C08630=1208.864,256.590,-63.182,-176.980,6.754,148.359
C08631=1208.860,256.838,-63.209,-176.978,6.756,148.359
C08632=1208.855,257.087,-63.236,-176.975,6.759,148.359
C08633=1208.851,257.336,-63.263,-176.973,6.761,148.359
C08634=1208.847,257.584,-63.291,-176.970,6.763,148.358
C08635=1208.843,257.832,-63.317,-176.968,6.765,148.358
C08636=1208.838,258.081,-63.344,-176.965,6.768,148.358
C08637=1208.833,258.329,-63.371,-176.963,6.770,148.358
C08638=1208.829,258.578,-63.399,-176.960,6.772,148.358
C08639=1208.824,258.826,-63.426,-176.957,6.775,148.358
C08640=1208.820,259.075,-63.453,-176.955,6.776,148.357
C08641=1208.815,259.324,-63.480,-176.953,6.779,148.357
C08642=1208.811,259.572,-63.507,-176.950,6.781,148.357
C08643=1208.807,259.820,-63.534,-176.947,6.784,148.357
C08644=1208.802,260.068,-63.561,-176.945,6.785,148.357
C08645=1208.798,260.318,-63.589,-176.943,6.788,148.357
C08646=1208.794,260.566,-63.616,-176.939,6.790,148.356
C08647=1208.789,260.815,-63.643,-176.937,6.792,148.356
C08648=1208.785,261.062,-63.671,-176.935,6.794,148.356
C08649=1208.780,261.311,-63.698,-176.933,6.797,148.356
C08650=1208.776,261.560,-63.725,-176.929,6.799,148.356
C08651=1208.771,261.809,-63.752,-176.927,6.801,148.355
C08652=1208.767,262.057,-63.780,-176.925,6.803,148.355
C08653=1208.762,262.305,-63.807,-176.922,6.806,148.355
C08654=1208.758,262.554,-63.834,-176.919,6.808,148.355
C08655=1208.754,262.827,-63.864,-176.917,6.811,148.355
C08656=1208.748,263.099,-63.895,-176.914,6.813,148.354
C08657=1208.744,263.371,-63.924,-176.911,6.816,148.354
C08658=1208.739,263.644,-63.955,-176.908,6.819,148.354
C08659=1208.735,263.893,-63.982,-176.906,6.821,148.354
C08660=1208.730,264.141,-64.010,-176.903,6.823,148.354
C08661=1208.726,264.390,-64.037,-176.900,6.825,148.354
C08662=1208.721,264.638,-64.064,-176.898,6.828,148.353
C08663=1208.717,264.887,-64.092,-176.896,6.830,148.353
C08664=1208.712,265.135,-64.119,-176.893,6.833,148.353
C08665=1208.708,265.383,-64.147,-176.891,6.835,148.353
C08666=1208.704,265.632,-64.174,-176.888,6.837,148.353
C08667=1208.699,265.881,-64.201,-176.885,6.840,148.353
C08668=1208.695,266.129,-64.229,-176.883,6.841,148.352
C08669=1208.690,266.378,-64.257,-176.881,6.844,148.352
C08670=1208.686,266.626,-64.285,-176.877,6.846,148.352
C08671=1208.681,266.875,-64.312,-176.875,6.849,148.352
C08672=1208.677,267.122,-64.340,-176.873,6.851,148.352
C08673=1208.673,267.372,-64.367,-176.870,6.853,148.352
C08674=1208.669,267.620,-64.395,-176.868,6.856,148.352
C08675=1208.664,267.867,-64.423,-176.865,6.858,148.351
C08676=1208.660,268.117,-64.450,-176.862,6.861,148.351
C08677=1208.655,268.365,-64.479,-176.860,6.862,148.351
C08678=1208.650,268.613,-64.506,-176.858,6.865,148.351
C08679=1208.647,268.862,-64.534,-176.855,6.868,148.351
C08680=1208.642,269.110,-64.561,-176.852,6.869,148.350
C08681=1208.638,269.358,-64.589,-176.850,6.872,148.350
C08682=1208.634,269.607,-64.617,-176.847,6.874,148.350
C08683=1208.628,269.856,-64.644,-176.845,6.877,148.350
C08684=1208.624,270.103,-64.672,-176.843,6.879,148.350
C08685=1208.620,270.352,-64.700,-176.840,6.881,148.350
C08686=1208.616,270.601,-64.727,-176.838,6.884,148.350
C08687=1208.611,270.849,-64.756,-176.834,6.886,148.349
C08688=1208.607,271.097,-64.784,-176.832,6.889,148.349
C08689=1208.602,271.346,-64.811,-176.830,6.891,148.349
C08690=1208.598,271.594,-64.839,-176.827,6.893,148.349
C08691=1208.593,271.843,-64.868,-176.825,6.896,148.349
C08692=1208.590,272.091,-64.896,-176.822,6.897,148.349
C08693=1208.585,272.340,-64.923,-176.819,6.900,148.349
C08694=1208.581,272.588,-64.950,-176.817,6.903,148.349
C08695=1208.576,272.836,-64.979,-176.814,6.905,148.348
C08696=1208.572,273.084,-65.007,-176.812,6.908,148.348
C08697=1208.568,273.333,-65.035,-176.810,6.910,148.348
C08698=1208.563,273.582,-65.063,-176.807,6.912,148.348
C08699=1208.559,273.830,-65.091,-176.805,6.915,148.348
C08700=1208.555,274.078,-65.119,-176.802,6.917,148.347
C08701=1208.549,274.326,-65.147,-176.799,6.920,148.347
C08702=1208.546,274.575,-65.175,-176.797,6.922,148.347
C08703=1208.541,274.823,-65.203,-176.794,6.924,148.347
C08704=1208.537,275.072,-65.232,-176.792,6.927,148.347
C08705=1208.533,275.320,-65.260,-176.790,6.929,148.347
C08706=1208.528,275.569,-65.287,-176.787,6.932,148.347
C08707=1208.523,275.817,-65.315,-176.784,6.934,148.347
C08708=1208.520,276.065,-65.343,-176.782,6.937,148.347
C08709=1208.515,276.314,-65.372,-176.779,6.939,148.346
C08710=1208.511,276.562,-65.400,-176.777,6.941,148.346
C08711=1208.506,276.810,-65.428,-176.774,6.944,148.346
C08712=1208.502,277.059,-65.457,-176.772,6.946,148.346
C08713=1208.498,277.307,-65.484,-176.769,6.949,148.346
C08714=1208.493,277.556,-65.513,-176.767,6.951,148.346
C08715=1208.489,277.804,-65.541,-176.764,6.953,148.346
C08716=1208.484,278.053,-65.570,-176.762,6.956,148.345
C08717=1208.480,278.300,-65.597,-176.759,6.958,148.345
C08718=1208.476,278.549,-65.625,-176.756,6.961,148.345
C08719=1208.471,278.797,-65.655,-176.754,6.963,148.345
C08720=1208.468,279.045,-65.683,-176.751,6.966,148.345
C08721=1208.463,279.294,-65.711,-176.749,6.968,148.345
C08722=1208.459,279.542,-65.739,-176.747,6.970,148.345
C08723=1208.454,279.791,-65.768,-176.744,6.973,148.345
C08724=1208.450,280.039,-65.796,-176.742,6.975,148.345
C08725=1208.445,280.288,-65.824,-176.739,6.978,148.344
C08726=1208.441,280.535,-65.852,-176.737,6.980,148.344
C08727=1208.437,280.784,-65.882,-176.734,6.983,148.344
C08728=1208.432,281.033,-65.910,-176.731,6.985,148.344
C08729=1208.428,281.280,-65.938,-176.729,6.987,148.344
C08730=1208.424,281.529,-65.967,-176.726,6.990,148.344
C08731=1208.419,281.777,-65.995,-176.724,6.992,148.344
C08732=1208.415,282.025,-66.024,-176.721,6.995,148.344
C08733=1208.411,282.274,-66.052,-176.719,6.997,148.343
C08734=1208.406,282.522,-66.081,-176.716,7.000,148.343
C08735=1208.402,282.771,-66.109,-176.714,7.002,148.343
C08736=1208.398,283.018,-66.138,-176.712,7.004,148.343
C08737=1208.393,283.267,-66.167,-176.709,7.007,148.343
C08738=1208.389,283.516,-66.195,-176.707,7.010,148.343
C08739=1208.385,283.763,-66.224,-176.704,7.012,148.343
C08740=1208.380,284.012,-66.253,-176.701,7.014,148.343
C08741=1208.376,284.260,-66.280,-176.699,7.017,148.343
C08742=1208.372,284.508,-66.310,-176.697,7.020,148.343
C08743=1208.367,284.757,-66.339,-176.694,7.023,148.343
C08744=1208.363,285.005,-66.366,-176.691,7.025,148.342
C08745=1208.359,285.253,-66.396,-176.689,7.028,148.342
C08746=1208.354,285.502,-66.425,-176.687,7.030,148.342
C08747=1208.349,285.751,-66.453,-176.684,7.032,148.342
C08748=1208.346,285.999,-66.482,-176.681,7.035,148.342
C08749=1208.341,286.247,-66.511,-176.679,7.037,148.342
C08750=1208.336,286.495,-66.540,-176.676,7.040,148.342
C08751=1208.333,286.744,-66.568,-176.674,7.042,148.342
C08752=1208.328,286.992,-66.597,-176.671,7.045,148.341
C08753=1208.323,287.240,-66.626,-176.669,7.047,148.341
C08754=1208.319,287.488,-66.655,-176.666,7.050,148.341
C08755=1208.315,287.737,-66.683,-176.664,7.052,148.341
C08756=1208.311,287.985,-66.713,-176.661,7.055,148.341
C08757=1208.306,288.233,-66.741,-176.659,7.057,148.341
C08758=1208.302,288.482,-66.770,-176.656,7.060,148.341
C08759=1208.297,288.756,-66.802,-176.654,7.062,148.341
C08760=1208.292,289.030,-66.834,-176.651,7.065,148.341
C08761=1208.288,289.304,-66.866,-176.648,7.068,148.341
C08762=1208.283,289.578,-66.898,-176.646,7.071,148.341
C08763=1208.279,289.827,-66.927,-176.643,7.073,148.341
C08764=1208.274,290.076,-66.956,-176.641,7.076,148.341
C08765=1208.270,290.324,-66.985,-176.638,7.078,148.340
C08766=1208.265,290.572,-67.014,-176.635,7.081,148.340
C08767=1208.261,290.820,-67.043,-176.633,7.083,148.340
C08768=1208.257,291.068,-67.072,-176.631,7.086,148.340
C08769=1208.253,291.317,-67.101,-176.628,7.089,148.340
C08770=1208.248,291.565,-67.130,-176.626,7.092,148.340
C08771=1208.244,291.813,-67.159,-176.624,7.094,148.340
C08772=1208.240,292.061,-67.189,-176.621,7.097,148.340
C08773=1208.235,292.310,-67.218,-176.618,7.099,148.340
C08774=1208.231,292.558,-67.247,-176.616,7.102,148.340
C08775=1208.226,292.806,-67.276,-176.614,7.104,148.340
C08776=1208.222,293.054,-67.306,-176.611,7.107,148.340
C08777=1208.218,293.303,-67.334,-176.609,7.109,148.339
C08778=1208.214,293.551,-67.364,-176.606,7.112,148.339
C08779=1208.210,293.799,-67.393,-176.603,7.114,148.339
C08780=1208.206,294.048,-67.422,-176.601,7.117,148.339
C08781=1208.201,294.295,-67.451,-176.599,7.119,148.339
C08782=1208.197,294.544,-67.480,-176.596,7.122,148.339
C08783=1208.192,294.792,-67.509,-176.594,7.125,148.339
C08784=1208.188,295.041,-67.539,-176.591,7.128,148.339
C08785=1208.184,295.289,-67.568,-176.589,7.130,148.339
C08786=1208.180,295.537,-67.598,-176.586,7.133,148.339
C08787=1208.175,295.785,-67.627,-176.584,7.135,148.339
C08788=1208.171,296.033,-67.656,-176.581,7.138,148.339
C08789=1208.167,296.281,-67.686,-176.578,7.141,148.339
C08790=1208.163,296.529,-67.715,-176.576,7.143,148.339
C08791=1208.158,296.778,-67.744,-176.574,7.146,148.339
C08792=1208.153,297.027,-67.774,-176.571,7.148,148.338
C08793=1208.149,297.275,-67.803,-176.569,7.151,148.338
C08794=1208.145,297.523,-67.833,-176.567,7.153,148.338
C08795=1208.141,297.772,-67.862,-176.564,7.156,148.338
C08796=1208.136,298.019,-67.891,-176.562,7.159,148.338
C08797=1208.132,298.268,-67.921,-176.559,7.162,148.338
C08798=1208.127,298.516,-67.950,-176.557,7.164,148.338
C08799=1208.124,298.763,-67.980,-176.554,7.167,148.338
C08800=1208.119,299.012,-68.010,-176.552,7.169,148.338
C08801=1208.115,299.260,-68.039,-176.549,7.172,148.338
C08802=1208.111,299.508,-68.069,-176.547,7.174,148.338
C08803=1208.106,299.757,-68.099,-176.544,7.177,148.338
C08804=1208.102,300.005,-68.128,-176.542,7.179,148.338
C08805=1208.098,300.253,-68.158,-176.539,7.182,148.338
C08806=1208.094,300.502,-68.187,-176.537,7.185,148.338
C08807=1208.089,300.750,-68.217,-176.535,7.188,148.338
C08808=1208.085,300.998,-68.246,-176.532,7.191,148.338
C08809=1208.081,301.246,-68.277,-176.530,7.193,148.338
C08810=1208.076,301.494,-68.306,-176.527,7.196,148.338
C08811=1208.072,301.743,-68.336,-176.525,7.198,148.338
C08812=1208.068,301.991,-68.365,-176.522,7.201,148.338
C08813=1208.064,302.239,-68.395,-176.520,7.203,148.337
C08814=1208.059,302.486,-68.425,-176.517,7.206,148.337
C08815=1208.055,302.735,-68.455,-176.515,7.208,148.337
C08816=1208.050,302.983,-68.484,-176.513,7.211,148.337
C08817=1208.046,303.231,-68.513,-176.510,7.214,148.337
C08818=1208.042,303.479,-68.544,-176.508,7.217,148.337
C08819=1208.037,303.727,-68.574,-176.505,7.220,148.337
C08820=1208.033,303.976,-68.603,-176.503,7.222,148.337
C08821=1208.029,304.224,-68.634,-176.500,7.225,148.337
C08822=1208.025,304.473,-68.664,-176.498,7.227,148.337
C08823=1208.021,304.721,-68.693,-176.496,7.230,148.337
C08824=1208.017,304.969,-68.723,-176.493,7.232,148.337
C08825=1208.012,305.217,-68.753,-176.491,7.235,148.337
C08826=1208.008,305.465,-68.783,-176.489,7.239,148.337
C08827=1208.004,305.713,-68.813,-176.486,7.241,148.337
C08828=1207.999,305.962,-68.843,-176.484,7.244,148.337
C08829=1207.995,306.210,-68.872,-176.482,7.246,148.337
C08830=1207.990,306.458,-68.903,-176.479,7.249,148.337
C08831=1207.986,306.706,-68.933,-176.477,7.251,148.337
C08832=1207.982,306.954,-68.963,-176.474,7.254,148.337
C08833=1207.977,307.202,-68.993,-176.472,7.257,148.337
C08834=1207.973,307.450,-69.023,-176.469,7.260,148.337
C08835=1207.969,307.698,-69.053,-176.467,7.263,148.337
C08836=1207.965,307.946,-69.083,-176.464,7.265,148.337
C08837=1207.960,308.195,-69.113,-176.462,7.268,148.337
C08838=1207.956,308.442,-69.144,-176.460,7.270,148.337
C08839=1207.952,308.691,-69.173,-176.457,7.273,148.337
C08840=1207.948,308.939,-69.204,-176.455,7.276,148.337
C08841=1207.943,309.188,-69.234,-176.453,7.279,148.337
C08842=1207.940,309.435,-69.264,-176.450,7.282,148.337
C08843=1207.935,309.684,-69.294,-176.448,7.284,148.337
C08844=1207.931,309.932,-69.324,-176.445,7.287,148.337
C08845=1207.926,310.180,-69.355,-176.443,7.289,148.337
C08846=1207.922,310.428,-69.384,-176.440,7.292,148.337
C08847=1207.918,310.676,-69.415,-176.438,7.294,148.337
C08848=1207.914,310.925,-69.445,-176.436,7.298,148.337
C08849=1207.909,311.173,-69.476,-176.433,7.301,148.337
C08850=1207.905,311.420,-69.506,-176.431,7.303,148.337
C08851=1207.900,311.669,-69.536,-176.429,7.306,148.337
C08852=1207.896,311.917,-69.566,-176.426,7.308,148.337
C08853=1207.892,312.165,-69.597,-176.424,7.311,148.337
C08854=1207.889,312.413,-69.627,-176.422,7.315,148.337
C08855=1207.884,312.661,-69.657,-176.419,7.317,148.337
C08856=1207.879,312.909,-69.688,-176.417,7.320,148.337
C08857=1207.875,313.157,-69.718,-176.415,7.322,148.337
C08858=1207.871,313.405,-69.749,-176.412,7.325,148.337
C08859=1207.867,313.654,-69.779,-176.410,7.327,148.337
C08860=1207.862,313.902,-69.810,-176.408,7.331,148.337
C08861=1207.858,314.150,-69.840,-176.405,7.334,148.337
C08862=1207.854,314.398,-69.870,-176.403,7.336,148.337
C08863=1207.849,314.674,-69.904,-176.400,7.339,148.337
C08864=1207.844,314.950,-69.938,-176.397,7.342,148.337
C08865=1207.840,315.227,-69.972,-176.395,7.345,148.337
C08866=1207.835,315.503,-70.006,-176.393,7.348,148.337
C08867=1207.831,315.750,-70.037,-176.390,7.351,148.337
C08868=1207.826,315.998,-70.067,-176.388,7.353,148.337
C08869=1207.822,316.246,-70.098,-176.385,7.357,148.337
C08870=1207.818,316.495,-70.129,-176.383,7.360,148.337
C08871=1207.814,316.743,-70.159,-176.381,7.362,148.337
C08872=1207.810,316.991,-70.189,-176.378,7.365,148.337
C08873=1207.806,317.239,-70.220,-176.376,7.367,148.337
C08874=1207.801,317.487,-70.251,-176.374,7.371,148.338
C08875=1207.796,317.735,-70.282,-176.371,7.374,148.338
C08876=1207.792,317.983,-70.312,-176.369,7.376,148.338
C08877=1207.788,318.232,-70.343,-176.366,7.379,148.338
C08878=1207.784,318.480,-70.374,-176.365,7.381,148.338
C08879=1207.780,318.727,-70.404,-176.362,7.384,148.338
C08880=1207.776,318.976,-70.435,-176.359,7.387,148.338
C08881=1207.771,319.224,-70.466,-176.358,7.390,148.338
C08882=1207.767,319.472,-70.496,-176.355,7.393,148.338
C08883=1207.763,319.719,-70.527,-176.353,7.395,148.338
C08884=1207.759,319.968,-70.559,-176.350,7.398,148.338
C08885=1207.755,320.215,-70.589,-176.348,7.402,148.338
C08886=1207.750,320.463,-70.620,-176.346,7.404,148.338
C08887=1207.746,320.712,-70.651,-176.343,7.407,148.338
C08888=1207.742,320.960,-70.681,-176.341,7.409,148.338
C08889=1207.737,321.208,-70.712,-176.339,7.412,148.338
C08890=1207.733,321.456,-70.743,-176.336,7.415,148.338
C08891=1207.729,321.704,-70.775,-176.334,7.418,148.338
C08892=1207.725,321.952,-70.806,-176.332,7.421,148.338
C08893=1207.720,322.200,-70.837,-176.330,7.423,148.338
C08894=1207.717,322.448,-70.867,-176.327,7.427,148.338
C08895=1207.713,322.697,-70.898,-176.325,7.430,148.338
C08896=1207.708,322.944,-70.929,-176.323,7.432,148.339
C08897=1207.704,323.192,-70.960,-176.320,7.435,148.339
C08898=1207.700,323.441,-70.991,-176.318,7.437,148.339
C08899=1207.695,323.689,-71.022,-176.316,7.441,148.339
C08900=1207.691,323.937,-71.054,-176.313,7.444,148.339
C08901=1207.687,324.185,-71.085,-176.312,7.446,148.339
C08902=1207.683,324.432,-71.115,-176.309,7.449,148.339
C08903=1207.679,324.680,-71.147,-176.307,7.451,148.339
C08904=1207.675,324.928,-71.177,-176.305,7.455,148.339
C08905=1207.671,325.177,-71.209,-176.302,7.458,148.339
C08906=1207.666,325.424,-71.240,-176.300,7.460,148.339
C08907=1207.662,325.673,-71.271,-176.298,7.463,148.339
C08908=1207.658,325.921,-71.302,-176.296,7.466,148.339
C08909=1207.653,326.168,-71.333,-176.293,7.469,148.339
C08910=1207.649,326.417,-71.365,-176.291,7.472,148.339
C08911=1207.645,326.665,-71.395,-176.289,7.474,148.340
C08912=1207.641,326.913,-71.427,-176.286,7.478,148.340
C08913=1207.636,327.161,-71.458,-176.285,7.480,148.340
C08914=1207.633,327.409,-71.490,-176.282,7.483,148.340
C08915=1207.628,327.657,-71.521,-176.280,7.486,148.340
C08916=1207.624,327.905,-71.552,-176.278,7.489,148.340
C08917=1207.620,328.153,-71.583,-176.275,7.492,148.340
C08918=1207.615,328.400,-71.615,-176.273,7.494,148.340
C08919=1207.611,328.649,-71.646,-176.271,7.497,148.340
C08920=1207.607,328.896,-71.677,-176.268,7.501,148.340
C08921=1207.603,329.145,-71.708,-176.267,7.503,148.341
C08922=1207.599,329.392,-71.740,-176.264,7.506,148.341
C08923=1207.595,329.641,-71.771,-176.262,7.509,148.341
C08924=1207.590,329.888,-71.802,-176.260,7.512,148.341
C08925=1207.586,330.137,-71.834,-176.258,7.515,148.341
C08926=1207.581,330.384,-71.866,-176.255,7.517,148.341
C08927=1207.578,330.632,-71.897,-176.253,7.521,148.341
C08928=1207.573,330.880,-71.928,-176.251,7.524,148.341
C08929=1207.569,331.128,-71.960,-176.249,7.526,148.341
C08930=1207.565,331.376,-71.991,-176.247,7.529,148.342
C08931=1207.561,331.624,-72.023,-176.245,7.532,148.341
C08932=1207.557,331.872,-72.055,-176.242,7.535,148.342
C08933=1207.552,332.121,-72.086,-176.240,7.538,148.342
C08934=1207.548,332.369,-72.118,-176.238,7.541,148.342
C08935=1207.544,332.616,-72.149,-176.236,7.544,148.342
C08936=1207.540,332.864,-72.181,-176.234,7.546,148.342
C08937=1207.536,333.112,-72.212,-176.231,7.549,148.342
C08938=1207.532,333.360,-72.244,-176.229,7.552,148.342
C08939=1207.527,333.608,-72.276,-176.227,7.555,148.342
C08940=1207.523,333.856,-72.307,-176.225,7.558,148.343
C08941=1207.519,334.104,-72.339,-176.223,7.560,148.343
C08942=1207.515,334.352,-72.370,-176.221,7.564,148.343
C08943=1207.510,334.600,-72.403,-176.218,7.567,148.343
C08944=1207.506,334.847,-72.434,-176.216,7.569,148.343
C08945=1207.502,335.096,-72.465,-176.214,7.573,148.343
C08946=1207.498,335.344,-72.497,-176.212,7.575,148.343
C08947=1207.493,335.592,-72.529,-176.210,7.578,148.343
C08948=1207.490,335.840,-72.561,-176.208,7.582,148.344
C08949=1207.485,336.087,-72.593,-176.206,7.584,148.344
C08950=1207.482,336.335,-72.624,-176.203,7.587,148.344
C08951=1207.477,336.584,-72.657,-176.201,7.591,148.344
C08952=1207.473,336.832,-72.688,-176.199,7.593,148.344
C08953=1207.469,337.080,-72.719,-176.197,7.596,148.344
C08954=1207.464,337.328,-72.752,-176.195,7.599,148.344
C08955=1207.460,337.575,-72.783,-176.193,7.602,148.345
C08956=1207.456,337.823,-72.815,-176.191,7.605,148.345
C08957=1207.451,338.071,-72.847,-176.188,7.607,148.345
C08958=1207.448,338.319,-72.879,-176.186,7.611,148.345
C08959=1207.444,338.567,-72.911,-176.185,7.613,148.345
C08960=1207.439,338.815,-72.943,-176.182,7.617,148.345
C08961=1207.435,339.063,-72.975,-176.180,7.620,148.346
C08962=1207.431,339.311,-73.007,-176.178,7.622,148.346
C08963=1207.426,339.558,-73.039,-176.176,7.626,148.346
C08964=1207.423,339.806,-73.071,-176.174,7.628,148.346
C08965=1207.419,340.055,-73.102,-176.172,7.631,148.346
C08966=1207.415,340.303,-73.135,-176.170,7.634,148.346
C08967=1207.410,340.581,-73.171,-176.167,7.638,148.346
C08968=1207.405,340.858,-73.207,-176.165,7.641,148.347
C08969=1207.400,341.137,-73.243,-176.163,7.645,148.347
C08970=1207.395,341.415,-73.279,-176.160,7.648,148.347
C08971=1207.392,341.663,-73.311,-176.159,7.650,148.347
C08972=1207.387,341.911,-73.343,-176.156,7.653,148.347
C08973=1207.383,342.158,-73.375,-176.154,7.656,148.347
C08974=1207.380,342.406,-73.407,-176.152,7.659,148.348
C08975=1207.375,342.655,-73.440,-176.150,7.663,148.348
C08976=1207.371,342.902,-73.471,-176.148,7.665,148.348
C08977=1207.366,343.150,-73.503,-176.146,7.668,148.348
C08978=1207.363,343.398,-73.535,-176.144,7.671,148.349
C08979=1207.358,343.646,-73.568,-176.142,7.674,148.349
C08980=1207.354,343.894,-73.600,-176.140,7.678,148.349
C08981=1207.350,344.142,-73.632,-176.138,7.680,148.349
C08982=1207.345,344.390,-73.665,-176.136,7.683,148.349
C08983=1207.342,344.638,-73.697,-176.134,7.686,148.349
C08984=1207.337,344.885,-73.729,-176.132,7.689,148.350
C08985=1207.333,345.133,-73.761,-176.130,7.692,148.350
C08986=1207.329,345.382,-73.794,-176.128,7.695,148.350
C08987=1207.325,345.629,-73.826,-176.126,7.698,148.350
C08988=1207.320,345.877,-73.858,-176.124,7.701,148.350
C08989=1207.317,346.125,-73.890,-176.122,7.704,148.351
C08990=1207.312,346.373,-73.923,-176.120,7.707,148.351
C08991=1207.308,346.621,-73.956,-176.118,7.710,148.351
C08992=1207.304,346.869,-73.988,-176.116,7.712,148.351
C08993=1207.300,347.116,-74.020,-176.114,7.716,148.351
C08994=1207.296,347.364,-74.052,-176.112,7.719,148.352
C08995=1207.292,347.612,-74.085,-176.110,7.722,148.352
C08996=1207.287,347.860,-74.118,-176.108,7.725,148.352
C08997=1207.284,348.108,-74.150,-176.106,7.728,148.352
C08998=1207.279,348.355,-74.183,-176.104,7.731,148.352
C08999=1207.274,348.603,-74.215,-176.103,7.733,148.353
C09000=1207.271,348.851,-74.248,-176.100,7.737,148.353
C09001=1207.266,349.099,-74.280,-176.098,7.740,148.353
C09002=1207.262,349.347,-74.313,-176.097,7.743,148.353
C09003=1207.259,349.595,-74.345,-176.095,7.746,148.354
C09004=1207.255,349.843,-74.378,-176.093,7.749,148.354
C09005=1207.249,350.090,-74.410,-176.091,7.752,148.354
C09006=1207.246,350.338,-74.443,-176.089,7.755,148.354
C09007=1207.242,350.586,-74.475,-176.087,7.758,148.354
C09008=1207.237,350.834,-74.508,-176.085,7.761,148.355
C09009=1207.233,351.082,-74.541,-176.083,7.764,148.355
C09010=1207.230,351.330,-74.573,-176.081,7.767,148.355
C09011=1207.225,351.577,-74.607,-176.080,7.770,148.355
C09012=1207.221,351.826,-74.639,-176.078,7.773,148.356
C09013=1207.216,352.073,-74.672,-176.076,7.776,148.356
C09014=1207.213,352.321,-74.704,-176.074,7.779,148.356
C09015=1207.208,352.569,-74.737,-176.072,7.782,148.356
C09016=1207.204,352.816,-74.770,-176.070,7.785,148.357
C09017=1207.200,353.065,-74.802,-176.068,7.789,148.357
C09018=1207.196,353.312,-74.835,-176.066,7.791,148.357
C09019=1207.192,353.560,-74.868,-176.064,7.795,148.357
C09020=1207.188,353.808,-74.900,-176.063,7.797,148.358
C09021=1207.184,354.056,-74.934,-176.061,7.801,148.358
C09022=1207.180,354.304,-74.967,-176.059,7.803,148.358
C09023=1207.176,354.552,-74.999,-176.057,7.807,148.358
C09024=1207.172,354.799,-75.032,-176.056,7.809,148.359
C09025=1207.167,355.046,-75.065,-176.053,7.813,148.359
C09026=1207.163,355.294,-75.098,-176.052,7.815,148.359
C09027=1207.158,355.542,-75.130,-176.050,7.819,148.359
C09028=1207.154,355.790,-75.163,-176.048,7.821,148.360
C09029=1207.150,356.038,-75.197,-176.046,7.825,148.360
C09030=1207.147,356.285,-75.229,-176.044,7.828,148.360
C09031=1207.143,356.533,-75.262,-176.043,7.831,148.361
C09032=1207.138,356.781,-75.295,-176.041,7.834,148.361
C09033=1207.134,357.029,-75.328,-176.039,7.837,148.361
C09034=1207.130,357.277,-75.361,-176.037,7.840,148.362
C09035=1207.126,357.525,-75.394,-176.035,7.843,148.362
C09036=1207.122,357.772,-75.427,-176.034,7.847,148.362
C09037=1207.118,358.020,-75.460,-176.032,7.849,148.362
C09038=1207.113,358.268,-75.494,-176.030,7.852,148.363
C09039=1207.110,358.516,-75.525,-176.029,7.855,148.363
C09040=1207.106,358.764,-75.559,-176.026,7.859,148.363
C09041=1207.101,359.011,-75.592,-176.025,7.861,148.364
C09042=1207.097,359.259,-75.625,-176.023,7.865,148.364
C09043=1207.093,359.507,-75.658,-176.022,7.867,148.364
C09044=1207.089,359.754,-75.691,-176.020,7.871,148.364
C09045=1207.085,360.002,-75.724,-176.018,7.873,148.365
C09046=1207.081,360.250,-75.758,-176.016,7.877,148.365
C09047=1207.077,360.498,-75.791,-176.015,7.880,148.365
C09048=1207.072,360.745,-75.824,-176.013,7.883,148.366
C09049=1207.068,360.993,-75.857,-176.011,7.886,148.366
C09050=1207.065,361.242,-75.891,-176.009,7.889,148.366
C09051=1207.061,361.489,-75.924,-176.008,7.892,148.367
C09052=1207.056,361.737,-75.957,-176.006,7.895,148.367
C09053=1207.052,361.985,-75.990,-176.005,7.898,148.367
C09054=1207.048,362.232,-76.023,-176.003,7.901,148.367
C09055=1207.044,362.480,-76.056,-176.001,7.904,148.368
C09056=1207.040,362.728,-76.089,-176.000,7.907,148.368
C09057=1207.036,362.975,-76.123,-175.998,7.911,148.369
C09058=1207.032,363.223,-76.156,-175.997,7.913,148.369
C09059=1207.028,363.470,-76.190,-175.994,7.917,148.369
C09060=1207.024,363.718,-76.223,-175.993,7.920,148.370
C09061=1207.019,363.966,-76.257,-175.992,7.923,148.370
C09062=1207.015,364.214,-76.290,-175.990,7.926,148.370
C09063=1207.011,364.462,-76.323,-175.989,7.929,148.371
C09064=1207.007,364.710,-76.356,-175.987,7.932,148.371
C09065=1207.003,364.957,-76.390,-175.985,7.935,148.371
C09066=1206.999,365.205,-76.423,-175.983,7.938,148.372
C09067=1206.995,365.453,-76.457,-175.982,7.941,148.372
C09068=1206.991,365.700,-76.490,-175.981,7.944,148.372
C09069=1206.987,365.948,-76.523,-175.979,7.947,148.373
C09070=1206.983,366.195,-76.557,-175.978,7.950,148.373
C09071=1206.978,366.477,-76.595,-175.976,7.954,148.373
C09072=1206.974,366.757,-76.632,-175.974,7.957,148.374
C09073=1206.969,367.037,-76.671,-175.972,7.961,148.374
C09074=1206.964,367.317,-76.708,-175.971,7.964,148.375
C09075=1206.960,367.565,-76.742,-175.969,7.967,148.375
C09076=1206.956,367.813,-76.776,-175.968,7.970,148.375
C09077=1206.952,368.061,-76.810,-175.967,7.973,148.376
C09078=1206.948,368.308,-76.843,-175.965,7.976,148.376
C09079=1206.944,368.556,-76.876,-175.964,7.979,148.377
C09080=1206.939,368.804,-76.910,-175.962,7.982,148.377
C09081=1206.935,369.051,-76.944,-175.960,7.985,148.377
C09082=1206.932,369.300,-76.977,-175.959,7.988,148.378
C09083=1206.928,369.547,-77.011,-175.958,7.991,148.378
C09084=1206.924,369.794,-77.044,-175.957,7.994,148.378
C09085=1206.919,370.042,-77.078,-175.955,7.998,148.379
C09086=1206.915,370.290,-77.112,-175.954,8.000,148.379
C09087=1206.911,370.537,-77.145,-175.952,8.003,148.380
C09088=1206.907,370.786,-77.178,-175.951,8.007,148.380
C09089=1206.903,371.033,-77.213,-175.949,8.010,148.380
C09090=1206.899,371.281,-77.246,-175.948,8.012,148.381
C09091=1206.895,371.528,-77.280,-175.947,8.015,148.381
C09092=1206.890,371.776,-77.314,-175.945,8.019,148.382
C09093=1206.887,372.024,-77.348,-175.944,8.022,148.382
C09094=1206.882,372.272,-77.381,-175.943,8.024,148.382
C09095=1206.879,372.519,-77.415,-175.942,8.027,148.383
C09096=1206.874,372.767,-77.449,-175.940,8.030,148.383
C09097=1206.871,373.015,-77.483,-175.939,8.034,148.384
C09098=1206.866,373.262,-77.516,-175.937,8.037,148.384
C09099=1206.862,373.510,-77.550,-175.936,8.039,148.384
C09100=1206.858,373.757,-77.584,-175.935,8.042,148.385
C09101=1206.854,374.005,-77.618,-175.934,8.045,148.385
C09102=1206.850,374.253,-77.652,-175.932,8.049,148.386
C09103=1206.846,374.500,-77.686,-175.931,8.051,148.386
C09104=1206.842,374.748,-77.719,-175.930,8.054,148.386
C09105=1206.838,374.996,-77.753,-175.929,8.057,148.387
C09106=1206.834,375.243,-77.787,-175.928,8.060,148.387
C09107=1206.830,375.491,-77.821,-175.926,8.063,148.388
C09108=1206.825,375.739,-77.855,-175.925,8.066,148.388
C09109=1206.822,375.987,-77.889,-175.924,8.069,148.389
C09110=1206.817,376.234,-77.923,-175.922,8.072,148.389
C09111=1206.813,376.481,-77.957,-175.922,8.075,148.390
C09112=1206.809,376.729,-77.990,-175.920,8.078,148.390
C09113=1206.805,376.977,-78.025,-175.919,8.081,148.390
C09114=1206.801,377.224,-78.059,-175.918,8.084,148.391
C09115=1206.796,377.472,-78.092,-175.917,8.087,148.391
C09116=1206.793,377.720,-78.127,-175.916,8.090,148.392
C09117=1206.789,377.967,-78.161,-175.915,8.092,148.392
C09118=1206.784,378.215,-78.194,-175.914,8.095,148.393
C09119=1206.781,378.463,-78.228,-175.912,8.098,148.393
C09120=1206.777,378.711,-78.263,-175.912,8.101,148.394
C09121=1206.772,378.958,-78.296,-175.910,8.104,148.394
C09122=1206.768,379.206,-78.331,-175.909,8.107,148.394
C09123=1206.765,379.454,-78.365,-175.908,8.110,148.395
C09124=1206.760,379.701,-78.399,-175.907,8.113,148.395
C09125=1206.756,379.949,-78.433,-175.906,8.116,148.396
C09126=1206.752,380.197,-78.467,-175.905,8.119,148.396
C09127=1206.748,380.444,-78.501,-175.904,8.121,148.397
C09128=1206.744,380.691,-78.535,-175.903,8.124,148.397
C09129=1206.740,380.940,-78.569,-175.902,8.127,148.398
C09130=1206.736,381.187,-78.603,-175.901,8.130,148.398
C09131=1206.732,381.434,-78.638,-175.900,8.133,148.399
C09132=1206.728,381.682,-78.672,-175.899,8.136,148.399
C09133=1206.724,381.930,-78.706,-175.898,8.139,148.399
